FUNCTION "SSA_Analog_S5_to_S7" : VOID	// FC 109
TITLE = Scale S7 Analogues for S5
//COPYRIGHT:    (C) 1998 BY  BUHLER AG
//                           CH-9240 UZWIL  SWITZERLAND
//
//PRODUCT:      AME01_98
//
//TITLE:        Scale S7 Analogues for S5
//              
//
//-------------------------------------------------------------------------
//
//IDENT:        AUTHOR:             DEPT:             DATE:
//
//FC109.1A      GS                  CDDP              15-Jan-2000
//              1st Release
//
//-------------------------------------------------------------------------
//
//PURPOSE: 
//
//RESTRICTIONS: 
//
//-------------------------------------------------------------------------
//
//Functions
//=========
//
//AI_Type:
//   1= S5 Analogue Input 4..20mA
//   2= S5 Analogue Input 0..+-10V or 0.. +-20mA
//   3= S5 Analogue Input PT100
// 
//  11= S5 Analogue Output 4..20mA
//  12= S5 Analogue Output 0..+-10V or 0.. +-20mA
AUTHOR : GS
FAMILY : ASW
NAME : ANA_S5_S
VERSION : 1.0
VAR_INPUT
  AI_Type : INT ;	//S5 Signal:
END_VAR
VAR_TEMP
  Inputvalue : INT ;
  OutputValue : INT ;
END_VAR
BEGIN
NETWORK
TITLE = Initialisation
      TAK;
      T     #Inputvalue;
NETWORK
TITLE = S5 Analogue Input 4..20mA
// (network holds code this reader does not know; not shown)
// S5 Analogue inputs cards 4..20mA give a number of 0..2560
// but have an offset of 512. This gives 512..2560 = 4..20mA
// 2048 units cover 16mA.
// Bottom 3 bits are used for over/under range indication from the card
// All S7 modules use 0..27648 as 0..100%
// Conversion formula is:-
//  
//     (S5Value - 512)  * 27648
//     ---------------
//          2048
// 
NETWORK
TITLE = S5 Analogue Input: 0..+-10V , 0..+-20mA
// (network holds code this reader does not know; not shown)
// S5 Analogue inputs cards 0..20mA give a number of 0..2048
// Bottom 3 bits are used for over/under range indication from the card
// All S7 modules use 0..27648 as 0..100%
// Conversion formula is:-
//  
//     S5Value  * 27648
//     -------
//      2048
// 
NETWORK
TITLE = S5 Analogue Input: PT100
// (network holds code this reader does not know; not shown)
// S5 Analogue inputs cards 0..20mA give a number of 0..2048
// Bottom 3 bits are used for over/under range indication from the card
// All S7 modules use 0..27648 as 0..100%
// Conversion formula is:-
//  
//     (S5Value-1024)  * 27648
//     -------
//      1024
// 
NETWORK
TITLE = S5 Analogue Output 4..20mA
      L     #AI_Type;
      L     11;
      <>I;
      JC    M007;
// S5 Analogue Outputs cards use a number of 0..1024
// Bottom 4 bits are not used used
// All S7 modules use 0..27648 as 0..100%
// Conversion formula is:-
//  
//    ( S7Value  * 820 ) + 204
//      -------
//       27648
// 
// Note:   820 is 4/5ths of 1024    (for the 4..20mA portion)
//         204 is 1/5th of 1024     (for the 0..4mA portion)
// 
      L     #Inputvalue;
      DTR;
      L     2.764800e+04;	// 27648
      /R;
      L     8.200000e+02;	// 820
      *R;
      L     2.040000e+02;	// 204
      +R;
      RND;
      SLW   4;
      T     #OutputValue;
M007: NOP   0;
NETWORK
TITLE = S5 Analogue Output 0..20mA or 4..20mA card
      L     #AI_Type;
      L     12;
      <>I;
      JC    M008;
// S5 Analogue Outputs cards use a number of 0..1024
// Bottom 4 bits are not used used
// All S7 modules use 0..27648 as 0..100%
// Conversion formula is:-
//  
//     S7Value  * 1024
//     -------
//      27648
// 
      L     #Inputvalue;
      DTR;
      L     2.764800e+04;	// 27648
      /R;
      L     1.024000e+03;	// 1024
      *R;
      RND;
      SLW   4;
      T     #OutputValue;
M008: NOP   0;
NETWORK
TITLE = Output final value
      L     #OutputValue;
END_FUNCTION

FUNCTION "STD_LineSecStdSub" : VOID	// FC 120
TITLE = Line and section control standard subroutines
//COPYRIGHT:    (C) 2000 BY  BUHLER LTD.
//                           CH-9240 UZWIL  SWITZERLAND
//
//PRODUCT:      STD_MU664    
//
//TITLE:        Line and section control standard subroutines
//              
//              Standardfunktionen für Linien und Sektionen              
//              
//
//--------------------------------------------------------------------------------
//
//IDENT:        AUTOR:              DEPT:                              DATE:
//STD_FC120.2.0 A.Egli              CT3                                18-Oct-2002
//              - New release
//STD_FC120.1.12Ph. Engler          MU664                              23-Aug-2002
//              - Function (4,1) added: Search group manual mode
//STD_FC120.1.11Ph. Engler          MU664                              30-Apr-2002
//              - Function (1,55) and (2,55) modified: Stopping/Stopped
//STD_FC120.1.10Ph. Engler          MU664                              21-Mar-2002
//              - Function (2,55): starting until S.ToSSW.infStarted
//STD_FC120.1.9 Ph. Engler          MU664                              12-Mar-2002
//              Status codes for WinCoS implemented:
//              - General group colour code
//              - Line and Section info code
//STD_FC120.1.8 Ph. Engler          MU664                              20-Mar-2001
//              Line status colour for 2-4 section implemented
//STD_FC120.1.7 Ph. Engler          MU664                              20-Dec-2000
//              Pre stop weight for cmdSequenceStop
//STD_FC120.1.6 Ph. Engler          MU664                              14-Dec-2000
//              - Substitude Bincode into recipe extended, InCode 3 
//              - JS Job paramter flags (2,2) Sta-Address corrected
//STD_FC120.1.5 Ph. Engler          MU664                              01-Nov-2000
//              CmdSequenceStop only if section is in StActive           
//STD_FC120.1.4 Ph. Engler          MU664                              19-Okt-2000
//              Update SND-Binlist staSameSndRcv:
//               Suppression of the error meassage 'bin not found'
//STD_FC120.1.3 Ph. Engler          MU664                              28-Jun-2000
//              Section text and colour code extension 
//              with code 702, 703 and 1402
//STD_FC120.1.2 Ph. Engler          MU664                              04-May-2000
//              LS Line state/fault protocolling (1,10)
//               esXXX corrected 
//STD_FC120.1.1 Ph. Engler          MU664                              29-Mar-2000
//              Line log messages implemented
//STD_FC120.1.0 Ph. Engler          MU664                              05-Jan-2000
//              1st Release
//
//--------------------------------------------------------------------------------
//
//PURPOSE:      These function are callt by Line Control and
//              Section Control.
//              The most subroutine are handled by FB90
//
//RESTRICTIONS:
//
//--------------------------------------------------------------------------------
//
//InCode: 
//1000 to 1999: Subroutines Line
//              For Input and Output parameter is 
//              LineDB.VarTemp used  
//2000 to 2999: Subroutines Section
//              For Input and Output parameter is
//              SectionDB.VarTemp used  
//
//
//
//
AUTHOR : PE
FAMILY : STD
VERSION : 2.0
VAR_INPUT
  InCode : INT ;	//Code number; 1000=Line 2=Section
END_VAR
BEGIN
NETWORK
TITLE = Input Data
NETWORK
TITLE = Sub1031: CF Clear line flags 
//Open DB=  Line Parameter DB
      L     #InCode;
      L     1031;
      <>I;
      JC    CF00;
//Line parameter DB
      L     L#0;
      T     DBD 140;	// Section 1
      T     DBD 144;	// Section 2
      T     DBD 148;	// Section 3
      T     DBD 152;	// Section 4
      T     DBD 156;	// General
      T     DBD 160;	// General
CF00: NOP   0;
NETWORK
TITLE = All other Subroutines are handled by FB90
      CDB;
      L     #InCode;
      T     DIW 0;	//InCode
//Call Methode FB90
      UC    "STD_LineSecStdSub2";
END_FUNCTION

FUNCTION "ASW_StageCtrl_Fct" : VOID	// FC 1800
TITLE = Scale Control: Main routines
//COPYRIGHT:    (C) 1994 BY  BUHLER LTD.
//                           CH-9240 UZWIL  SWITZERLAND
//
//PRODUCT:      GCS7
//
//TITLE:        Stage Control
//
//Revision: 10
//
//-------------------------------------------------------------------------
//
//IDENT:        AUTOR:              DEPT:                         DATE:
//
//FC1800.1A     A.Egli              BSAE                          12.02.2008
//              Convert from S5 Version 2F
//
//-------------------------------------------------------------------------
//
//PURPOSE:      
//
//RESTRICTIONS:
//
//-------------------------------------------------------------------------
//
//FC-PARAMETER:
//------------
//InCode:
//
//   2= Init Batch
//   6= Next Stage
//
//  12= Init Stage
//      Update Stage.ScaleUsed
//      Stage.ScaleStarted:=0
//      Stage.ScaleDone
//
//
//  
AUTHOR : EA
FAMILY : GCS7UL
NAME : SCC_MAN
VERSION : 3.3
VAR_INPUT
  InCode : INT ;	// CODE
  Stage : UDT 18000;
END_VAR
VAR_TEMP
  tmpScaleDB : INT ;
  tmpScaleNr : DINT ;
  tmpScaleBit : DINT ;
  tmpRecipePlace : INT ;
  tmpRecipeDB : INT ;
  tmpRecipeAddrIngr : DINT ;
  tmpSecDB : INT ;
  tmpAddStage : DINT ;
  ConstMaxStage : INT ;
  tmpIdx : INT ;
  tmpOffsetIngr : INT ;	//Offest 1st Ingedient Stage [BYTE]
  tmpBinNo : INT ;
  tmpArrayIdxScale : INT ;
END_VAR
BEGIN
NETWORK
TITLE =
      L     2;
      T     #ConstMaxStage;
NETWORK
TITLE =
      L     P##Stage;
      LAR1;
      L     W [AR1,P#0.0];
      T     #tmpSecDB;
      L     D [AR1,P#2.0];
      T     #tmpAddStage;
NETWORK
TITLE = Call Section DB
      OPN   DB [#tmpSecDB];
      L     DBW 230;	// "SecDB".JobAc.RecipePlace
      T     #tmpRecipePlace;
NETWORK
TITLE = Methode 2: Init Batch
      L     #InCode;
      L     2;
      <>I;
      JC    iEnd;
      L     1;
      BLD   5;
      T     LD 36;	//--> Init Stage
      TAK;
      T     LD 40;
      L     P##Stage;
      LAR1;
      L     W [AR1,P#0.0];
      T     LW 34;
      OPN   DB [LW 34];
      L     D [AR1,P#2.0];
      LAR1;
      L     LD 40;
      L     LD 36;
      T     W [AR1,P#4.0];
      JU    dJ0;
iEnd: NOP   0;
NETWORK
TITLE = Methode 6: Next Stage
      L     #InCode;
      L     2;
      <>I;
      JC    nEnd;
      BLD   5;
      T     LD 36;
      TAK;
      T     LD 40;
      L     P##Stage;
      LAR1;
      L     W [AR1,P#0.0];
      T     LW 34;
      OPN   DB [LW 34];
      L     D [AR1,P#2.0];
      LAR1;
      L     LD 40;	//--> Init Stage
      L     LD 36;
      AN     [AR1,P#0.1];
      BLD   5;
      T     LD 36;
      TAK;
      T     LD 40;
      L     P##Stage;
      LAR1;
      L     W [AR1,P#0.0];
      T     LW 34;
      OPN   DB [LW 34];
      L     D [AR1,P#2.0];
      LAR1;
      L     LD 40;
      L     LD 36;
      AN     [AR1,P#2.0];
      BEC;
      L     #ConstMaxStage;
      BLD   5;
      T     LD 36;
      TAK;
      T     LD 40;
      L     P##Stage;
      LAR1;
      L     W [AR1,P#0.0];
      T     LW 34;
      OPN   DB [LW 34];
      L     D [AR1,P#2.0];
      LAR1;
      L     LD 40;
      L     LD 36;
      L     W [AR1,P#4.0];
      ==I;
      BLD   5;
      T     LD 36;
      TAK;
      T     LD 40;
      L     P##Stage;
      LAR1;
      L     W [AR1,P#0.0];
      T     LW 34;
      OPN   DB [LW 34];
      L     D [AR1,P#2.0];
      LAR1;
      L     LD 40;
      L     LD 36;
      S      [AR1,P#2.1];
      BEC;
      BLD   5;
      T     LD 36;
      TAK;
      T     LD 40;
      L     P##Stage;
      LAR1;
      L     W [AR1,P#0.0];
      T     LW 34;
      OPN   DB [LW 34];
      L     D [AR1,P#2.0];
      LAR1;
      L     LD 40;
      L     LD 36;
      L     W [AR1,P#4.0];
      +     1;
      BLD   5;
      T     LD 36;
      TAK;
      T     LD 40;
      L     P##Stage;
      LAR1;
      L     W [AR1,P#0.0];
      T     LW 34;
      OPN   DB [LW 34];
      L     D [AR1,P#2.0];
      LAR1;
      L     LD 40;
      L     LD 36;
      T     W [AR1,P#4.0];
      JU    dJ0;
nEnd: NOP   0;
NETWORK
TITLE = Methode 12: Init Stage
//ACTUAL DB BY CALL: Line DB
      L     #InCode;
      L     1;
      <>I;
      JC    dEnd;
//--------------------
//Init 
dJ0:  LAR1  #tmpAddStage;
      L     0;
      T     DBD [AR1,P#10.0];	//Stage.ScaleUsed
      T     DBD [AR1,P#14.0];	//Stage.ScaleUsed
      L     0;
      T     DBD [AR1,P#18.0];	//Stage.ScaleStarted
      T     DBD [AR1,P#22.0];	//Stage.ScaleStarted
      L     0;
      T     DBD [AR1,P#26.0];	//Stage.ScaleDone
      T     DBD [AR1,P#30.0];	//Stage.ScaleDone
      SET;
      BLD   5;
      T     LD 36;
      TAK;
      T     LD 40;
//Test Stage Number
      L     P##Stage;
      LAR1;
      L     W [AR1,P#0.0];
      T     LW 34;
      OPN   DB [LW 34];
      L     D [AR1,P#2.0];
      LAR1;
      L     LD 40;
//--------------------
//Loop over all In reipe used scales
      L     LD 36;
      R      [AR1,P#0.1];	//  
      BLD   5;
      T     LD 36;
      TAK;
      T     LD 40;	// "SecDB".JobNom.ScaleUsed[x]
      L     P##Stage;
      LAR1;
      L     W [AR1,P#0.0];
      T     LW 34;	//--> DB8.ScaleNr
      OPN   DB [LW 34];	// Subroutine ScalePointer
      L     D [AR1,P#2.0];
      LAR1;	//<--DB8.ScaleDB
      L     LD 40;
      L     LD 36;	// No Scale
      R      [AR1,P#0.0];
      BLD   5;
//--------------------
//Calculate Pointer to CWA Recipe
      T     LD 36;	// >>> CALL Scale-DB
      TAK;
      T     LD 40;
      L     P##Stage;
      LAR1;	// REC .ParNrOfIngrPerRecipe
      L     W [AR1,P#0.0];
      T     LW 34;
      OPN   DB [LW 34];
      L     D [AR1,P#2.0];
      LAR1;	// SCDB.ParNrOfBytePerIngr
      L     LD 40;	// 
      L     LD 36;	//---> Offset 1st Ingr. actual Stage
      R      [AR1,P#2.1];	// REC .ParNrOfIngrPerRecipe
      BLD   5;	// SCDB.ParNrOfBytePerIngr
      T     LD 36;	// 
      TAK;
      T     LD 40;	// 
      L     P##Stage;	// REC.ParDwNrFirstRecipe
      LAR1;	// --> Start Recipe[x]
      L     W [AR1,P#0.0];
      T     LW 34;
      OPN   DB [LW 34];
      L     D [AR1,P#2.0];	//-->Address Ingrediewnt 
      LAR1;
      L     LD 40;	// REC.ParDBNrRecipe
      L     LD 36;
//--------------------
//Read Ingredient from CWA recipe
      S      [AR1,P#2.0];	// >>> CALL Scale-DB
      BLD   5;
      T     LD 36;
//--------------------
//Set Scale Used
      TAK;
      T     LD 40;
      L     P##Stage;
      LAR1;	//--> not used
      L     W [AR1,P#0.0];
      T     LW 34;
      OPN   DB [LW 34];
      L     D [AR1,P#2.0];	//Stage.ScaleUsedStage
      LAR1;
      L     LD 40;
      L     LD 36;
      L     W [AR1,P#4.0];
      L     0;
//---------------------------------
//Test Stage Empty
      ==I;
      JC    dSta;
      BLD   5;
      T     LD 36;
      TAK;
      T     LD 40;
      L     P##Stage;
      LAR1;
      L     W [AR1,P#0.0];
      T     LW 34;
// -- END LOOP SCALE -----------
      OPN   DB [LW 34];
      L     D [AR1,P#2.0];
      LAR1;
      L     LD 40;
      L     LD 36;
      L     W [AR1,P#4.0];
      L     #ConstMaxStage;
      >I;
      JC    dSta;
      L     1;
dLPS: T     #tmpScaleNr;
      +     -1;
      T     #tmpArrayIdxScale;
      LAR1;
      AN    DBX [AR1,P#170.0];
      JC    dNxt;
      OPN   DI 8;
      L     #tmpScaleNr;
      T     DIW 20;
      CALL  "GCS7_ScaleCtrlSub" (
           CODE                     := 3);
      L     DIW 22;
      T     #tmpScaleDB;
      L     0;
      ==I;
      JC    dNxt;
      OPN   DI [#tmpScaleDB];
      BLD   5;
      T     LD 36;
      TAK;
      T     LD 40;
      L     P##Stage;
      LAR1;
      L     W [AR1,P#0.0];
      T     LW 34;
      OPN   DB [LW 34];
      L     D [AR1,P#2.0];
      LAR1;
      L     LD 40;
      L     LD 36;
      L     W [AR1,P#4.0];
      +     -1;
      T     #tmpIdx;
      L     DIW 104;
      L     #ConstMaxStage;
      /I;
      L     #tmpIdx;
      *I;
      L     DIW 106;
      *I;
      T     #tmpOffsetIngr;
      L     DIW 104;
      L     DIW 106;
      *I;
      L     #tmpRecipePlace;
      *I;
      L     DIW 100;
      +I;
      L     #tmpOffsetIngr;
      +D;
      SLD   3;
      T     #tmpRecipeAddrIngr;
      LAR1;
      L     DIW 98;
      T     #tmpRecipeDB;
      OPN   DI [#tmpRecipeDB];
      L     DIW [#tmpRecipeAddrIngr];
      T     #tmpBinNo;
      L     #tmpBinNo;
      L     0;
      ==I;
      JC    dNxt;
      LAR1  #tmpAddStage;
      L     #tmpArrayIdxScale;
      +AR1;
      S     DBX [AR1,P#10.0];
dNxt: L     64;
      L     #tmpScaleNr;
      +     1;
      >I;
      JC    dLPS;
dSta: LAR1  #tmpAddStage;
      L     DBD [AR1,P#10.0];
      L     0;
      ==D;
      A(;
      L     DBD [AR1,P#14.0];
      L     0;
      ==D;
      );
      BLD   5;
      T     LD 36;
      TAK;
      T     LD 40;
      L     P##Stage;
      LAR1;
      L     W [AR1,P#0.0];
      T     LW 34;
      OPN   DB [LW 34];
      L     D [AR1,P#2.0];
      LAR1;
      L     LD 40;
      L     LD 36;
      =      [AR1,P#2.0];
      BEU;
dEnd: NOP   0;
END_FUNCTION

FUNCTION "SSA_Vis_Update" : VOID	// FC 2042
TITLE = SSA_VIS_Status
//
//COPYRIGHT:    (C) 1996  BUHLER AG, CH-9240 UZWIL, SWITZERLAND
//
//PRODUCT:      SSA_VIS_Hsk
//
//TITLE:        Update hanshake bits for graphik update
//
//REVISION:     0
//-------------------------------------------------------------------------
//
//IDENT:        AUTHOR:             DEPT:                       DATE:
//FC2043.1.0    A. Egli             CT3                         19-Dec-2007
//              1st Release in S7
//
//-------------------------------------------------------------------------
//
//PURPOSE:      MANUAL : 
//
//RESTRICTIONS: S7
//-------------------------------------------------------------------------
//
FAMILY : ASW
NAME : SSA_VIS
VERSION : 1.0
VAR_INPUT
  HskDB : BLOCK_DB ;	//Pointer to Object Status
END_VAR
BEGIN
NETWORK
TITLE = Read Pointer
      OPN   #HskDB;
NETWORK
TITLE = Reset Handshake Bits
      NOP   0;
// Set Handshake Bit
      L     DBD 66;	// PCWrite_Graphic_Hsk
      INVD;	// 
      L     DBD 48;	// PCRead_Graphic_Hsk
      AD;	//  
      L     DBD 30;	// Graphic_Refresh
      OD;	// 
      T     DBD 48;	// PCRead_Graphic_Hsk
      L     DBD 70;	// PCWrite_Graphic_Hsk
      INVD;	// 
      L     DBD 52;	// PCRead_Graphic_Hsk
      AD;	//  
      L     DBD 34;	// Graphic_Refresh
      OD;	// 
      T     DBD 52;	// PCRead_Graphic_Hsk
      L     DBW 74;	// PCWrite_Graphic_Hsk
      INVI;	// 
      L     DBW 56;	// PCRead_Graphic_Hsk
      AW;	//  
      L     DBW 38;	// Graphic_Refresh
      OW;	// 
      T     DBW 56;	// PCRead_Graphic_Hsk
// Nachfrischen loeschen
      L     DBD 66;	//PCWrite_Graphic_Hsk
      INVD;
      L     DBD 30;	//Graphic_Refresh 
      AD;
      T     DBD 30;	//Graphic_Refresh
      L     DBD 70;	//PCWrite_Graphic_Hsk
      INVD;
      L     DBD 34;	//Graphic_Refresh 
      AD;
      T     DBD 34;	//Graphic_Refresh
      L     DBW 74;	//PCWrite_Graphic_Hsk
      INVI;
      L     DBW 38;	//Graphic_Refresh 
      AW;
      T     DBW 38;	//Graphic_Refresh
// Loeschen HS-Bit von VISCONTROL
      L     0;
      T     DBD 66;	//PCWrite_Graphic_Hsk
      T     DBD 70;	//PCWrite_Graphic_Hsk
      T     DBW 74;	//PCWrite_Graphic_Hsk
END_FUNCTION

FUNCTION "SSA_VIS_Status" : VOID	// FC 2043
TITLE = SSA_VIS_Status
//
//COPYRIGHT:    (C) 1996  BUHLER AG, CH-9240 UZWIL, SWITZERLAND
//
//PRODUCT:      SSA_VIS_Status
//
//TITLE:        Convert Status for Viscontrol
//
//REVISION:     0
//-------------------------------------------------------------------------
//
//IDENT:        AUTHOR:             DEPT:                       DATE:
//FC2043.1.0    A. Egli             CT3                         19-Dec-2007
//              1st Release in S7
//
//-------------------------------------------------------------------------
//
//PURPOSE:      MANUAL : 
//
//RESTRICTIONS: S7
//-------------------------------------------------------------------------
//
FAMILY : ASW
NAME : SSA_VIS
VERSION : 1.0
VAR_INPUT
  InObject : POINTER ;	//Pointer to Object Status
  OType : INT ;	//Object Type
  OutVisStatus : POINTER ;	//Pointer to Viscontrol Status in Picture DB
END_VAR
VAR_TEMP
  SrcDB : INT ;
  SrcAddress : DINT ;
  DstDB : INT ;
  DstAddress : DINT ;
  tmpDX : INT ;
END_VAR
BEGIN
NETWORK
TITLE = Read Pointer
      L     P##InObject;
      LAR1;
      L     W [AR1,P#0.0];
      T     #SrcDB;
      L     D [AR1,P#2.0];
      T     #SrcAddress;
      LAR2;
      OPN   DI [#SrcDB];
      L     P##OutVisStatus;
      LAR1;
      L     W [AR1,P#0.0];
      T     #DstDB;
      L     D [AR1,P#2.0];
      T     #DstAddress;
NETWORK
TITLE = Check Object Type
      L     1300;
      L     #OType;
      >=I;
      JC    ElMa;	//Element
      L     2300;
      L     #OType;
      >=I;
      JC    ElMa;	//Machine
      L     3000;
      L     #OType;
      ==I;
      JC    Gr;
      BEU;
NETWORK
TITLE =
ElMa: L     1000;
      /I;
      SRD   16;
      T     #tmpDX;
      JU    Calc;
NETWORK
TITLE =
Gr:   LAR2  P#DIX 0.0;
      A     DIX [AR2,P#21.4];	//Gr.OutWarning
      O     DIX [AR2,P#17.4];	//Gr.StFault
      L     2;
      JC    TRAN;
      O     DIX [AR2,P#17.2];	//Gr.StStarted
      O     DIX [AR2,P#17.3];	//Gr.StStopping
      L     1;
      JC    TRAN;
      O     DIX [AR2,P#17.0];	//Gr.StStopped
      O     DIX [AR2,P#17.1];	//Gr.StStarting
      L     0;
      JC    TRAN;
      L     99;
      JU    TRAN;
NETWORK
TITLE = Convert Status of ELement or Machine with Filter DB
Calc: NOP   0;
      L     123;
      L     #tmpDX;
      >I;
      JC    Err;
      L     249;
      L     #tmpDX;
      <I;
      JC    Err;
      +     -123;
      L     P#16.0;
      *D;
      L     P#20.0;
      +D;
      LAR1;
      OPN   "SSA_VIS_Filter";
//----------------------
//Test First Left Bytes without Status
      L     DBD [AR1,P#12.0];	//STATUS = 3
      L     DW#16#FFFFFF00;
      AD;
      L     DID [AR2,P#2.0];
      AD;
      JZ    STL2;
      L     3;
      JU    TRAN;
STL2: L     DBD [AR1,P#8.0];	//STATUS = 2
      L     DW#16#FFFFFF00;
      AD;
      L     DID [AR2,P#2.0];
      AD;
      JZ    STL1;
      L     2;
      JU    TRAN;
STL1: L     DBD [AR1,P#4.0];	//STATUS = 1
      L     DW#16#FFFFFF00;
      AD;
      L     DID [AR2,P#2.0];
      AD;
      JZ    STL0;
      L     1;
      JU    TRAN;
STL0: L     DBD [AR1,P#0.0];
      L     DW#16#FFFFFF00;
      AD;
      L     DID [AR2,P#2.0];
      AD;
      JZ    STR3;
      L     0;
      JU    TRAN;
//----------------------
//Test Right Bytes with Status
STR3: L     DBD [AR1,P#12.0];	//STATUS = 3
      L     DW#16#FF;
      AD;
      L     DID [AR2,P#2.0];
      AD;
      JZ    STR2;
      L     3;
      JU    TRAN;
STR2: L     DBD [AR1,P#8.0];	//STATUS = 2
      L     DW#16#FF;
      AD;
      L     DID [AR2,P#2.0];
      AD;
      JZ    STR1;
      L     2;
      JU    TRAN;
STR1: L     DBD [AR1,P#4.0];	//STATUS = 1
      L     DW#16#FF;
      AD;
      L     DID [AR2,P#2.0];
      AD;
      JZ    STR0;
      L     1;
      JU    TRAN;
STR0: L     DBD [AR1,P#0.0];	//STATUS = 0
      L     DW#16#FF;
      AD;
      L     DID [AR2,P#2.0];
      AD;
      JZ    Err;
      L     0;
      JU    TRAN;
Err:  L     99;	//Error
NETWORK
TITLE = Write Status to Picture DB
TRAN: OPN   DB [#DstDB];
      LAR1  #DstAddress;
      L     DBW [AR1,P#0.0];
      TAK;
      ==I;
      T     DBW [AR1,P#0.0];
      BEC;
//Set Change Bit
      L     #DstAddress;
      L     DW#16#FFFFF;
      AD;
      SRD   3;
      +     -2;
      L     "SSA_VIS_Filter".ParBlockLen;
      /I;
      L     2#1;
      SLW;
      OPN   DB [#DstDB];
      L     DBB 1;
      OW;
      T     DBB 1;
END_FUNCTION

FUNCTION "SSA_VIS_Log_Msg" : VOID	// FC 2055
TITLE = SSA_VIS_Log_Msg
//
//COPYRIGHT:    (C) 1996  BUHLER AG, CH-9240 UZWIL, SWITZERLAND
//
//PRODUCT:      GCS7R1
//
//TITLE:        LOG-TRANSFER FROM QUEUE TO VIS-VONTROL HANDSHAKE-DB
//
//REVISION:     0
//-------------------------------------------------------------------------
//
//IDENT:        AUTHOR:             DEPT:                       DATE:
//FC2055.1.0    A. Egli             CT3                         19-Dec-2007
//              1st Release in S7
//
//-------------------------------------------------------------------------
//
//PURPOSE:      MANUAL : 
//
//RESTRICTIONS: S7
//-------------------------------------------------------------------------
//
FAMILY : ASW
NAME : SSA_VIS
VERSION : 1.0
VAR_INPUT
  HSDB : BLOCK_DB ;	//VISCONTROL-HANDSHAKE-DB
  LogQueue : BLOCK_DB ;	//LOG-WARTESCHLANGE
  PCNr : INT ;	//UNTERSTUETZT WERDEN 2 PC's PCNR=1 und PCNR=2
  VDU : BOOL ;	//BITINFORMATION, OB VDU-MELDUNG ODER NICHT
END_VAR
VAR_TEMP
  tmpPC1 : BOOL ;
  tmpPC2 : BOOL ;
END_VAR
BEGIN
NETWORK
TITLE = Init
      L     #PCNr;
      L     1;
      ==I;
      =     #tmpPC1;	//PC 1
      L     #PCNr;
      L     2;
      ==I;
      =     #tmpPC2;	//PC 2
NETWORK
TITLE =
      OPN   #LogQueue;
      CDB;
      OPN   #HSDB;
NETWORK
TITLE = Reset Handshake LOG
      OPN   #HSDB;	// AUFRUF HSDB
      L     DBW 76;	// HSDB.PCWrite_LOG_Hsk   :  VIS->PLC:LOG-Daten gelesen
      INVI;	// 
      L     DBW 58;	// HSDB.PCRead_LOG_Hsk
      AW;
      T     DBW 58;	// HSDB.PCRead_LOG_Hsk    :  Reset Handshake Bits to PC
      L     0;
      T     DBW 76;	// HSDB.PCWrite_LOG_Hsk   :  Reset Handshake Bits from PC
NETWORK
TITLE = Enter Next Message
      AN    DIX 57.0;	//LogDB.HskPLCtoPC.PC1
      A     #tmpPC1;	//PC 1
      O;
      AN    DIX 57.1;	//LogDB.HskPLCtoPC.PC2
      A     #tmpPC2;	//PC 2
      O;
      A     DBX 59.0;	//HskDB.PCRead_LOG_Hsk 
      AN    #VDU;	//)  Element-Meldungen
      O;
      A     DBX 59.1;	//HskDB.PCRead_LOG_Hsk
      A     #VDU;	// VDU-Meldungen
      JC    END;
//Enter Next Message
      AN    #VDU;	// Element-Meldung
      JC    LOG;
      L     DIB 64;
      T     DBW 102;	// HskDB.Bildnummer
      S     DBX 59.1;	// HskDB.PCRead_LOG_Hsk.Bildnummer gueltig
      JU    RESE;
LOG:  L     DIW 60;	//)
      L     2#11111;	// )  LOG-HEAD KLASSE = 0
      AW;	// )
      L     16;	//)
      >=I;
      L     DIW 60;	// )
      JC    CWA;	// )
      L     2#1111111100011111;	// )  LOG-HEAD KLASSE = 0
      AW;	//  )
CWA:  T     DBW 78;	//-->HskDB.PCReadLog
      L     DIW 62;	// LogDB.PC.Msg[1]
      T     DBW 80;	//-->HskDB.PCReadLog
      L     DID 64;	// LogDB.PC.Msg[1]
      T     DBD 82;	//-->HskDB.PCReadLog
      L     DID 68;	// LogDB.PC.Msg[1]
      T     DBD 86;	//-->HskDB.PCReadLog
      L     DID 72;	// LogDB.PC.Msg[1]
      T     DBD 90;	//-->HskDB.PCReadLog
      L     DID 76;	// LogDB.PC.Msg[1]
      T     DBD 94;	//-->HskDB.PCReadLog
      L     DID 80;	// LogDB.PC.Msg[1]
      T     DBD 98;	//-->HskDB.PCReadLog
      SET;
      =     DBX 59.0;	//HskDB.PCRead_LOG_Hsk: Neue LOG-Daten!
//Set Message Done
RESE: A     #tmpPC1;	//PC1
      S     DIX 49.0;	//LogDB.PC.HskPC1toPLC 
      A     #tmpPC2;	//PC2
      S     DIX 51.0;	//LogDB.PC.HskPC2toPLC
END:  NOP   0;
END_FUNCTION

DATA_BLOCK "SYS_CBitDB"	// DB 2
TITLE = SYS: Changebit interface
//COPYRIGHT:    (C) 1994 BY  BUHLER LTD.
//                           CH-9240 UZWIL  SWITZERLAND
//
//PRODUCT:      GCS90
//
//TITLE:        Change-DB
//
//-------------------------------------------------------------------------
//
//IDENT:        AUTOR:              DEPT:                         DATE:
//
//DB250.1A      A.Egli              AEE61                         08-Jul-96
//                 1st Release
//
//-------------------------------------------------------------------------
//
//PURPOSE:      MANUAL : CBITMAN
//              CODE   : FB 74
//
//RESTRICTIONS:
//
//-------------------------------------------------------------------------
//
//$EJECT
//
//
//
//
AUTHOR : EA
FAMILY : GCS7SYS
NAME : CBIT_DB
VERSION : 0.0
  STRUCT
   Spare0 : WORD ;
   Spare2 : WORD ;
   Spare4 : WORD ;
   ParNextDB : INT ;	//Next Change-Bit DB
   Spare8 : WORD ;
   ParDWCopyBits : INT  := 512;	//Byte address of Copy[1]
   ParBlockLen : INT  := 120;	//Length datablock per change bit
   Spare14 : WORD ;
   Spare16 : WORD ;
   Spare18 : WORD ;
   VarTemp : ARRAY  [1 .. 10 ] OF //Working memory
   WORD ;
   RBit : ARRAY  [1 .. 1280 ] OF //-- PC Write ---------
   BOOL ;
   CBIT : ARRAY  [1 .. 1280 ] OF //-- PC Read  ------------
   BOOL ;
   Value : ARRAY  [1 .. 76 ] OF //Fast value for PC
   INT ;
   Copy : ARRAY  [1 .. 1280 ] OF //Internal used
   BOOL ;
   ParPointer : STRUCT 	//-- Configuaration source address --
    B001 : STRUCT
     DBNr : INT ;
     DWNr : INT ;
    END_STRUCT ;
    B005 : STRUCT
     DBNr : INT ;
     DWNr : INT ;
    END_STRUCT ;
    B009 : STRUCT
     DBNr : INT ;
     DWNr : INT ;
    END_STRUCT ;
    B013 : STRUCT
     DBNr : INT ;
     DWNr : INT ;
    END_STRUCT ;
    B017 : STRUCT
     DBNr : INT ;
     DWNr : INT ;
    END_STRUCT ;
    B021 : STRUCT
     DBNr : INT ;
     DWNr : INT ;
    END_STRUCT ;
    B025 : STRUCT
     DBNr : INT ;
     DWNr : INT ;
    END_STRUCT ;
    B029 : STRUCT
     DBNr : INT ;
     DWNr : INT ;
    END_STRUCT ;
    B033 : STRUCT
     DBNr : INT ;
     DWNr : INT ;
    END_STRUCT ;
    B037 : STRUCT
     DBNr : INT ;
     DWNr : INT ;
    END_STRUCT ;
    B041 : STRUCT
     DBNr : INT ;
     DWNr : INT ;
    END_STRUCT ;
    B045 : STRUCT
     DBNr : INT ;
     DWNr : INT ;
    END_STRUCT ;
    B049 : STRUCT
     DBNr : INT ;
     DWNr : INT ;
    END_STRUCT ;
    B053 : STRUCT
     DBNr : INT ;
     DWNr : INT ;
    END_STRUCT ;
    B057 : STRUCT
     DBNr : INT ;
     DWNr : INT ;
    END_STRUCT ;
    B061 : STRUCT
     DBNr : INT ;
     DWNr : INT ;
    END_STRUCT ;
    B065 : STRUCT
     DBNr : INT ;
     DWNr : INT ;
    END_STRUCT ;
    B069 : STRUCT
     DBNr : INT ;
     DWNr : INT ;
    END_STRUCT ;
    B073 : STRUCT
     DBNr : INT ;
     DWNr : INT ;
    END_STRUCT ;
    B077 : STRUCT
     DBNr : INT ;
     DWNr : INT ;
    END_STRUCT ;
    B081 : STRUCT
     DBNr : INT ;
     DWNr : INT ;
    END_STRUCT ;
    B085 : STRUCT
     DBNr : INT ;
     DWNr : INT ;
    END_STRUCT ;
    B089 : STRUCT
     DBNr : INT ;
     DWNr : INT ;
    END_STRUCT ;
    B093 : STRUCT
     DBNr : INT ;
     DWNr : INT ;
    END_STRUCT ;
    B097 : STRUCT
     DBNr : INT ;
     DWNr : INT ;
    END_STRUCT ;
    B101 : STRUCT
     DBNr : INT ;
     DWNr : INT ;
    END_STRUCT ;
    B105 : STRUCT
     DBNr : INT ;
     DWNr : INT ;
    END_STRUCT ;
    B109 : STRUCT
     DBNr : INT ;
     DWNr : INT ;
    END_STRUCT ;
    B113 : STRUCT
     DBNr : INT ;
     DWNr : INT ;
    END_STRUCT ;
    B117 : STRUCT
     DBNr : INT ;
     DWNr : INT ;
    END_STRUCT ;
    B121 : STRUCT
     DBNr : INT ;
     DWNr : INT ;
    END_STRUCT ;
   END_STRUCT ;
  END_STRUCT ;	
BEGIN
   ParDWCopyBits := 512;
   ParBlockLen := 120;
   ParPointer.B001.DBNr := -1;
END_DATA_BLOCK

DATA_BLOCK "SYS_DirectCtrlDB"	// DB 3
TITLE = GCS7: PC direct control interface default DB
AUTHOR : EA
FAMILY : GCS7SYS
NAME : PCCtrl
VERSION : 0.0
  STRUCT
   Spare0 : WORD ;
   Spare2 : WORD ;
   Spare4 : WORD ;
   Spare6 : DWORD ;
   Spare10 : DWORD ;
   ParAnswerTime : INT  := 5;	//Maximum time for answer
   VarActControlDB : INT ;	//DB from actual communication
   VarAnswerTime : INT ;	//Actual answer time
   GC : STRUCT 	//=== Working memory
    InDBNr : INT ;
    InDynLen : INT ;
    InDynAddr : DINT ;
    InParaLen : INT ;
    InParaAddr : DINT ;
    Revision : INT ;
    Temp8 : DINT ;
   END_STRUCT ;
   ChangeBit : STRUCT 	//Change Bit
    Spare : BYTE ;
    CBit1 : BOOL ;	//Function done
    CBit2 : BOOL ;
    CBit3 : BOOL ;
    CBit4 : BOOL ;
   END_STRUCT ;
   PC : STRUCT 	//== PC: Read/Write
    Hsk : STRUCT 	// Handshake
     Spare0 : BYTE ;
     FDefineCmd : BOOL ;
     FDefinePara : BOOL ;
     FDefineValue : BOOL ;
     FExamine : BOOL ;
     F04 : BOOL ;
     F05 : BOOL ;
     F06 : BOOL ;
     F07 : BOOL ;
    END_STRUCT ;
    ErrObj : INT ;	//Spare
    ErrCode : INT ;	//Fault reason: 0=No Fault
    ObjectType : INT ;	//Type of addressed object
    ObjectNo : INT ;	//Addressd object
    Cmd1 : ARRAY  [0 .. 15 ] OF BOOL ;
    Cmd2 : ARRAY  [0 .. 15 ] OF BOOL ;
    Cmd3 : ARRAY  [0 .. 15 ] OF BOOL ;
    Value : ARRAY  [1 .. 100 ] OF //Data from or for actual object
    WORD ;
   END_STRUCT ;
  END_STRUCT ;	
BEGIN
   ParAnswerTime := 5;
END_DATA_BLOCK

DATA_BLOCK "SYS_HornDB"	// DB 4
TITLE = GCS7: Data Horn Modul
//COPYRIGHT:    (C) 2000 BUHLER AG, CH-9240 UZWIL, SWITZERLAND
//                           
//PRODUCT:      Horn DB
//              Horn DB
//
//TITLE:        Horn Modul
//              
//
//--------------------------------------------------------------------------------
//
//IDENT:        AUTHOR:             DEPT:                              DATE:
//
//P01_DB004.2.0 A_Egli              CT3                                29.Okt.2002
//              1st Release
//
//-------------------------------------------------------------------------
//
AUTHOR : EA
FAMILY : GCSS7
NAME : HornDB
VERSION : 2.0
  STRUCT
   All : STRUCT
    CmdHornOff : BOOL ;
    Spare1 : BOOL ;
    Spare2 : BOOL ;
    Spare3 : BOOL ;
    Spare4 : BOOL ;
    Spare5 : BOOL ;
   END_STRUCT ;
   _1_A901Horn : STRUCT
    CmdHornOff : BOOL ;
    CmdHornOn : BOOL ;
    StartWarning : BOOL ;
    Spare1 : BOOL ;
    Spare2 : BOOL ;
   END_STRUCT ;
   _1_A902Horn : STRUCT
    CmdHornOff : BOOL ;
    CmdHornOn : BOOL ;
    StartWarning : BOOL ;
    Spare1 : BOOL ;
    Spare2 : BOOL ;
   END_STRUCT ;
   _1_A903Horn : STRUCT
    CmdHornOff : BOOL ;
    CmdHornOn : BOOL ;
    StartWarning : BOOL ;
    Spare1 : BOOL ;
    Spare2 : BOOL ;
   END_STRUCT ;
   _1_A904Horn : STRUCT
    CmdHornOff : BOOL ;
    CmdHornOn : BOOL ;
    StartWarning : BOOL ;
    Spare1 : BOOL ;
    Spare2 : BOOL ;
   END_STRUCT ;
  END_STRUCT ;	
BEGIN
END_DATA_BLOCK

DATA_BLOCK "SYS_LOG_Queue"	// DB 5
TITLE = SYS_LOG_Queue
//COPYRIGHT:    (C) 1996 BY  BUHLER LTD.
//                           CH-9240 UZWIL  SWITZERLAND
//
//PRODUCT:      GCS90_OS.LOG
//
//TITLE:        QUEUE-DB
//
//-------------------------------------------------------------------------
//
//IDENT:        AUTOR:              DEPT:                       DATE:
//
//DB5.1A        S. Kalberer         AEE61                       4-Jun-1996
//              1st Release in S7, converted from DB220.1A
//
//-------------------------------------------------------------------------
//
//PURPOSE:      MANUAL : LOGMAN
//              CODE   : FB46,47
//
//RESTRICTIONS: S7
//              only for PC-Interface
//
//-------------------------------------------------------------------------
//
//
AUTHOR : SK
FAMILY : GCS7SYS
NAME : LOG_DB
VERSION : 0.0
  STRUCT
   spare0 : WORD ;
   ParByteStartQueue : INT  := 180;	//1st Byte of ParMsgQueue
   spare4 : INT ;
   ParMaxNoOfMsg : INT  := 100;	//Max index of array MsgQueue
   VarNrOfMsgInQueue : INT ;	//Actual number of Msg in queue
   VarByteWrite : INT ;	//Write pointer
   VarByteRead : INT ;	//Read pointer
   ParByteMsgFull : INT  := 156;	//1st Byte or ParMsgFull
   varMsg : STRUCT 	//== Working memory
    Header : WORD ;
    Para1 : WORD ;
    Para2 : WORD ;
    Para3 : WORD ;
    Para4 : WORD ;
    Para5 : WORD ;
    Para6 : WORD ;
    Para7 : WORD ;
    Para8 : WORD ;
    Para9 : WORD ;
    Para10 : WORD ;
    Para11 : WORD ;
   END_STRUCT ;
   ChangeBit : STRUCT
    spare : BYTE ;
    CBit0 : BOOL ;
   END_STRUCT ;
   ParNrOfMsgMemory : INT  := 1;	//Max index of array PC.Msg
   spare : BYTE ;
   ParPC1Connected : BOOL  := TRUE;	//Pc1 is connected
   ParPC2Connected : BOOL ;	//Pc1 is connected
   ParPC3Connected : BOOL ;	//Pc1 is connected
   ParPC4Connected : BOOL ;	//Pc1 is connected
   spare4504 : BOOL ;
   spare4505 : BOOL ;
   spare4506 : BOOL ;
   spare4507 : BOOL ;
   spare4600 : BOOL ;
   spare4601 : BOOL ;
   spare4602 : BOOL ;
   spare4603 : BOOL ;
   spare4604 : BOOL ;
   spare4605 : BOOL ;
   CmdAddFastMsg : BOOL ;	//->Add Fast Message directly at PC interface
   CmdResetLog : BOOL  := TRUE;	//->Init Queue
   InPC1Online : BOOL ;	//->PC1 is offline
   InPC2Online : BOOL ;	//->PC2 is offline
   InPC3Online : BOOL ;	//->PC3 is offline
   InPC4Online : BOOL ;	//->PC4 is offline
   PC : STRUCT 	//=== Interface to PC
    HskPC1toPLC : WORD ;
    HskPC2toPLC : WORD ;
    HskPC3toPLC : WORD ;
    HskPC4toPLC : WORD ;
    HskPLCtoPC : WORD ;
    NrOfMessageInQueue : WORD ;
    Msg : ARRAY  [1 .. 4 ] OF //Message for PC
    STRUCT
     Header : WORD ;
     Para1 : WORD ;
     Para2 : WORD ;
     Para3 : WORD ;
     Para4 : WORD ;
     Para5 : WORD ;
     Para6 : WORD ;
     Para7 : WORD ;
     Para8 : WORD ;
     Para9 : WORD ;
     Para10 : WORD ;
     Para11 : WORD ;
    END_STRUCT ;
   END_STRUCT ;
   ParMsgFull : STRUCT 	//===Message queue full
    Header : WORD  := W#16#8C;
    Para1 : WORD ;
    Para2 : WORD ;
    Para3 : WORD ;
    Para4 : WORD ;
    Para5 : WORD ;
    Para6 : WORD ;
    Para7 : WORD ;
    Para8 : WORD ;
    Para9 : WORD ;
    Para10 : WORD ;
    Para11 : WORD  := W#16#B;
   END_STRUCT ;
   MsgQueue : ARRAY  [1 .. 100 ] OF //=== Message buffer =========
   STRUCT
    Header : WORD ;
    Para1 : WORD ;
    Para2 : WORD ;
    Para3 : WORD ;
    Para4 : WORD ;
    Para5 : WORD ;
    Para6 : WORD ;
    Para7 : WORD ;
    Para8 : WORD ;
    Para9 : WORD ;
    Para10 : WORD ;
    Para11 : WORD ;
   END_STRUCT ;
  END_STRUCT ;	
BEGIN
   ParByteStartQueue := 180;
   ParMaxNoOfMsg := 100;
   ParByteMsgFull := 156;
   ParNrOfMsgMemory := 1;
   ParPC1Connected := TRUE;
   CmdResetLog := TRUE;
   ParMsgFull.Header := W#16#8C;
   ParMsgFull.Para11 := W#16#B;
END_DATA_BLOCK

DATA_BLOCK "GCS7_GrCtrlDBTmp"	// DB 6
AUTHOR : EA
FAMILY : GCS7UL
VERSION : 0.0
"GCS7_GrpCtrlMain"
BEGIN
END_DATA_BLOCK

DATA_BLOCK "GCS7_ScaleControlDB"	// DB 8
TITLE = GCS7_ScaleControlDB: Data of Scale Control modul
//
//COPYRIGHT:    (C) 1994 BY  BUHLER LTD.
//                           CH-9240 UZWIL  SWITZERLAND
//
//PRODUCT:      GCS90
//
//TITLE:        SCALE-CONTROL
//
//-------------------------------------------------------------------------
//
//IDENT:       AUTOR:              DEPT:             DATE:
//
//DB8.1A        A_Egli              AEE61             21.11.96
//              1st Release
//
//-------------------------------------------------------------------------
//
//PURPOSE:      MANUAL : SCCMAN
//              CODE   : FC68/FC69...
//
//RESTRICTIONS:
//
//-------------------------------------------------------------------------
//
//
AUTHOR : EA
FAMILY : GCS90UL
NAME : SCC_DB
VERSION : 0.0
  STRUCT
   spare0 : ARRAY  [0 .. 9 ] OF // reserved for parameter
   WORD ;
   VarTemp : ARRAY  [1 .. 11 ] OF // working memory
   WORD ;
   ParScaleDB : ARRAY  [1 .. 64 ] OF // Configuration of all scale DB
   INT ;
  END_STRUCT ;	
BEGIN
   ParScaleDB[1] := 201;
   ParScaleDB[2] := 202;
END_DATA_BLOCK

DATA_BLOCK "GCS7_GrCtrlDB"	// DB 9
TITLE = GCS7: Inteface Group to Group control
//COPYRIGHT:    (C) 2000 BUHLER AG, CH-9240 UZWIL, SWITZERLAND
//                           
//PRODUCT:      Gruppenverwaltung mit 320 Gruppen
//              Group Control with 320 groups
//
//TITLE:        Call Group FB
//              
//
//--------------------------------------------------------------------------------
//
//IDENT:        AUTHOR:             DEPT:                              DATE:
//
//P01_DB009.2.0 A_Egli              CT3                                31.Okt.2002
//              1st Release
//
//-------------------------------------------------------------------------
//
AUTHOR : EA
FAMILY : GCSS7
NAME : ObjDB
VERSION : 2.0
  STRUCT
   ParByteNoSecDB : INT  := 1012;	//Pointer to configuration of section DBs
   ParMaxGroupCnt : INT  := 10;	//1=32 Groups, 2=64 Groups,.. , 10= 320 Groups,
   OutManualAny : BOOL ;	//Any object of the plant in manual mode
   OutFaultAny : BOOL ;	//Any object of the plant has faull
   Spare4 : WORD ;
   Spare5 : WORD ;
   ParFeed : ARRAY  [1 .. 320 ] OF //Objects are feed groups
   BOOL ;
   ParMGR : ARRAY  [1 .. 320 ] OF //Objects are MGR
   BOOL ;
   ParWGR : ARRAY  [1 .. 320 ] OF //Objects are WGR
   BOOL ;
   ParGGR : ARRAY  [1 .. 320 ] OF //Objects are GGR
   BOOL ;
   ParShare : ARRAY  [1 .. 320 ] OF //Objects are possible to share
   BOOL ;
   OutShared : ARRAY  [1 .. 320 ] OF //Objects are shared at the moment
   BOOL ;
   OutOccupied : ARRAY  [1 .. 320 ] OF //Objects are occupied by any section
   BOOL ;
   OutEnable : ARRAY  [1 .. 320 ] OF //Enable for objects
   BOOL ;
   CmdNext : ARRAY  [1 .. 320 ] OF //Next command for objects
   BOOL ;
   CmdFaultReset : ARRAY  [1 .. 320 ] OF BOOL ;
   CmdManualOff : ARRAY  [1 .. 320 ] OF BOOL ;
   InStopped : ARRAY  [1 .. 320 ] OF BOOL ;
   InStarted : ARRAY  [1 .. 320 ] OF BOOL ;
   InFault : ARRAY  [1 .. 320 ] OF BOOL ;
   InWarning : ARRAY  [1 .. 320 ] OF BOOL ;
   InManual : ARRAY  [1 .. 320 ] OF BOOL ;
   InLocked : ARRAY  [1 .. 320 ] OF //Waiting until real group
   BOOL ;
   InExternal : ARRAY  [1 .. 320 ] OF //Is at the moment external used
   BOOL ;
   CmdContinue : ARRAY  [1 .. 320 ] OF //Is used as condition to set OutAutoStart
   BOOL ;
   InLoaded : ARRAY  [1 .. 320 ] OF //Group is loaded with product
   BOOL ;
   InDPFault : ARRAY  [1 .. 320 ] OF //Any element has DPFault
   BOOL ;
   InHWStop : ARRAY  [1 .. 320 ] OF //Any element has HWStop
   BOOL ;
   InAutoStart : ARRAY  [1 .. 320 ] OF //OutAutoStart is on
   BOOL ;
   InStartWarning : ARRAY  [1 .. 320 ] OF //InStartWarning is on
   BOOL ;
   OutConflictObj : ARRAY  [1 .. 320 ] OF BOOL ;
   OutConflictSecDB : INT ;
   Section : ARRAY  [1 .. 100 ] OF STRUCT
    DBNr : INT ;
    DBB : INT ;
   END_STRUCT ;
  END_STRUCT ;	
BEGIN
   ParByteNoSecDB := 1012;
   ParMaxGroupCnt := 10;
   ParFeed[26] := TRUE;
   ParFeed[33] := TRUE;
   ParFeed[41] := TRUE;
   ParFeed[43] := TRUE;
   ParFeed[46] := TRUE;
   ParMGR[22] := TRUE;
   ParMGR[24] := TRUE;
   ParMGR[31] := TRUE;
   ParMGR[32] := TRUE;
   ParMGR[42] := TRUE;
   ParMGR[44] := TRUE;
   ParMGR[45] := TRUE;
   ParMGR[47] := TRUE;
   ParMGR[196] := TRUE;
   ParWGR[12] := TRUE;
   ParWGR[13] := TRUE;
   ParWGR[21] := TRUE;
   ParWGR[23] := TRUE;
   ParWGR[28] := TRUE;
   ParGGR[1] := TRUE;
   ParGGR[2] := TRUE;
   ParGGR[7] := TRUE;
   ParShare[1] := TRUE;
   ParShare[2] := TRUE;
   ParShare[7] := TRUE;
END_DATA_BLOCK

DATA_BLOCK "SYS_DirectCtrlLCDB"	// DB 10
TITLE = GCS7: PC direct control interface default DB
AUTHOR : EA
FAMILY : GCS7SYS
NAME : PCCtrl
VERSION : 0.0
  STRUCT
   Spare0 : WORD ;
   Spare2 : WORD ;
   Spare4 : WORD ;
   Spare6 : DWORD ;
   Spare10 : DWORD ;
   ParAnswerTime : INT  := 10;	//Maximum time for answer
   VarActControlDB : INT ;	//DB from actual communication
   VarAnswerTime : INT ;	//Actual answer time
   GC : STRUCT 	//=== Working memory
    InDBNr : INT ;
    InDynLen : INT ;
    InDynAddr : DINT ;
    InParaLen : INT ;
    InParaAddr : DINT ;
    Set11Done : BOOL ;
    InObjectNo : INT ;
    InLCAddr : INT ;
   END_STRUCT ;
   ChangeBit : STRUCT 	//Change Bit
    Spare : BYTE ;
    CBit1 : BOOL ;	//Function done
    CBit2 : BOOL ;
    CBit3 : BOOL ;
    CBit4 : BOOL ;
   END_STRUCT ;
   PC : STRUCT 	//== PC: Read/Write
    Hsk : STRUCT 	// Handshake
     Spare0 : BYTE ;
     FDefineCmd : BOOL ;
     FDefinePara : BOOL ;
     FDefineValue : BOOL ;
     FExamine : BOOL ;
     FExamineFirst : BOOL ;
     FExamineNext : BOOL ;
     F06 : BOOL ;
     F07 : BOOL ;
    END_STRUCT ;
    ErrObj : INT ;	//Spare
    ErrCode : INT ;	//Fault reason: 0=No Fault
    ObjectType : INT ;	//Type of addressed object
    ObjectNo : INT ;	//Addressd object
    Cmd1 : ARRAY  [0 .. 15 ] OF BOOL ;
    Cmd2 : ARRAY  [0 .. 15 ] OF BOOL ;
    Cmd3 : ARRAY  [0 .. 15 ] OF BOOL ;
    Value : ARRAY  [1 .. 100 ] OF //Data from or for actual object
    WORD ;
   END_STRUCT ;
  END_STRUCT ;	
BEGIN
   ParAnswerTime := 10;
END_DATA_BLOCK

DATA_BLOCK "TEST_IOSimuliInput"	// DB 16
AUTHOR : EA
FAMILY : SIM
NAME : Inputs
VERSION : 0.1
  STRUCT
   in : ARRAY  [0 .. 1027 ] OF BYTE ;
  END_STRUCT ;	
BEGIN
END_DATA_BLOCK

DATA_BLOCK "TEST_IOSimuliOutput"	// DB 17
AUTHOR : EA
FAMILY : SIM
NAME : Inputs
VERSION : 0.1
  STRUCT
   in : ARRAY  [0 .. 1027 ] OF BYTE ;
  END_STRUCT ;	
BEGIN
END_DATA_BLOCK

DATA_BLOCK "KebaHT4Data"	// DB 20
AUTHOR : SK
FAMILY : KebaHT4
VERSION : 0.0
"KebaHT4"
BEGIN
END_DATA_BLOCK

DATA_BLOCK DB 21
TITLE = Reference List Motors for HT4 Control
//COPYRIGHT:    (C) 1999 BY  BUHLER LTD.
//                           CH-9240 UZWIL  SWITZERLAND
//
//PRODUCT:      
//
//TITLE:        REFERENCE LIST "MOTORS" FOR "MAINTENANCE MOTOR CONTROL HT4"
//
//              REFERENZLISTE "MOTOREN" FUER "LOKALE MOTOREN STEUERUNG HT4"
//
//---------------------------------------------------------------------------
//
//IDENT:        AUTHOR:              DEPT:                       DATE:
//
//DB81.1A       S. Kalberer          CT3                         14.04.1999
//              1st Release: adjusted from S5 DB181.2A
//
//---------------------------------------------------------------------------
//
//PURPOSE:      - REFERENCE TABLE FOR MOTOR ELEMENTS
//
//RESTRICTIONS: - S7
//              - THIS DB IS CALLED BY FB80.
//
//---------------------------------------------------------------------------
//
//STRUCTURE OF DB-BLOCKS:
//=======================
//Byte 00: DBW (WORD-Hex) = OBJECT No. (Motors with two direction/speed are marked with *)
//                                     (Motors with variable speed are marked with @)
//Byte 02: DBW (INT)  = Digital output 1 byte-address 
//Byte 04: DBW (INT)  = Digital output 1 bit-address
//Byte 06: DBW (INT)  = Digital output 2 byte-address 
//Byte 08: DBW (INT)  = Digital output 2 bit-address
//Byte 10: DBW (INT)  = Digital output 3 byte-address 
//Byte 12: DBW (INT)  = Digital output 3 bit-address
//Byte 14: DBW (INT)  = Digital output 4 byte-address 
//Byte 16: DBW (INT)  = Digital output 4 bit-address
//Byte 18: DBW (INT)  = Analog  output 1 address (byte)
//Byte 20: DBW (WORD) = Object  state
//
//PARAMETERS FOR OUTPUTS:
//=======================
//Motor: (with one direction or speed)
//DO_1 = Digital output address
//DO_2 = not used
//DO_3 = not used
//DO_4 = not used
//AO_1 = not used
//
//Motor: (with two directions or speed) *
//DO_1 = Digital output address (foreward/1.speed)
//DO_2 = Digital output address (reverse/2.speed)
//DO_3 = not used
//DO_4 = not used
//AO_1 = not used
//
//Motor: (with variable speed drive) @
//DO_1 = Digital output address
//DO_2 = not used
//DO_3 = not used
//DO_4 = not used
//AO_1 = Analog output address
//
//KNOW_HOW_PROTECT
// (falls angegeben, kann im generierten Baustein keine Änderungen mehr vorgenommen werden)
// (If specified, no more changes can be made once the block is generated)
//UNLINKED
// (falls angegeben, ist der generierte Baustein nur im AG Ladespeicher vorhanden) 
// (If specified, the generated block is only available in the PLC load memory)
//READ_ONLY
// (falls angegeben, ist der generierte Baustein im AG nicht änderbar)
// (If specified, the generated block cannot be changed in the programmable controller)
//
AUTHOR : ASW
FAMILY : Keba
NAME : DB_MOT
VERSION : 1.0
  STRUCT
   Obj : ARRAY  [1 .. 11 ] OF STRUCT
    No : WORD ;	//Object No. (e.g. 1002 for 1-M002)
    DO1_ByteAddr : INT ;	//DO1 (Byte Address)
    DO1_BitAddr : INT ;	//DO1 (Bit Address)
    DO2_ByteAddr : INT ;	//DO2 (Byte Address)
    DO2_BitAddr : INT ;	//DO2 (Bit Address)
    DO3_ByteAddr : INT ;	//DO3 (Byte Address)
    DO3_BitAddr : INT ;	//DO3 (Bit Address)
    DO4_ByteAddr : INT ;	//DO4 (Byte Address)
    DO4_BitAddr : INT ;	//DO4 (Bit Address)
    AO1_ByteAddr : INT ;	//AO1 (Byte Address)
    State : WORD ;	//State
   END_STRUCT ;
  END_STRUCT ;	
BEGIN
   Obj[1].No := W#16#1001;
   Obj[1].DO1_ByteAddr := 4;
   Obj[2].No := W#16#1002;
   Obj[2].DO1_ByteAddr := 4;
   Obj[2].DO1_BitAddr := 1;
   Obj[3].No := W#16#1003;
   Obj[3].DO1_ByteAddr := 4;
   Obj[3].DO1_BitAddr := 2;
   Obj[3].DO2_ByteAddr := 5;
   Obj[3].DO2_BitAddr := 2;
   Obj[4].No := W#16#1004;
   Obj[4].DO1_ByteAddr := 4;
   Obj[4].DO1_BitAddr := 3;
   Obj[4].DO2_ByteAddr := 5;
   Obj[4].DO2_BitAddr := 3;
   Obj[9].No := W#16#1010;
   Obj[9].DO1_ByteAddr := 4;
   Obj[9].DO1_BitAddr := 7;
   Obj[9].AO1_ByteAddr := 512;
   Obj[10].No := W#16#1011;
   Obj[10].DO1_ByteAddr := 5;
   Obj[10].AO1_ByteAddr := 20;
   Obj[11].No := W#16#FFFF;
END_DATA_BLOCK

DATA_BLOCK DB 22
TITLE = Reference List various Objects for HT4 Control
//COPYRIGHT:    (C) 1999 BY  BUHLER LTD.
//                           CH-9240 UZWIL  SWITZERLAND
//
//PRODUCT:      
//
//TITLE:        REFERENCE LIST "OBJECTS" FOR "MAINTENANCE MOTOR CONTROL HT4"
//
//              REFERENZLISTE "OBJEKTE" FUER "LOKALE MOTOREN STEUERUNG HT4"
//
//---------------------------------------------------------------------------
//
//IDENT:        AUTHOR:              DEPT:                       DATE:
//
//DB82.1A       S. Kalberer          CT3                         14.04.1999
//              1st Release: adjusted from S5 DB182.2A
//
//---------------------------------------------------------------------------
//
//PURPOSE:      - REFERENCE TABLE FOR VARIOUS ELEMENTS
//
//RESTRICTIONS: - S7
//              - THIS DB IS CALLED BY FB80.
//
//---------------------------------------------------------------------------
//
//STRUCTURE OF DB-BLOCKS:
//=======================
//Byte 00: DBW (WORD-Hex) = OBJECT No. (Motors with two direction/speed are marked with *)
//                                     (Motors with variable speed are marked with @)
//Byte 02: DBW (INT)  = Digital output 1 byte-address 
//Byte 04: DBW (INT)  = Digital output 1 bit-address
//Byte 06: DBW (INT)  = Digital output 2 byte-address 
//Byte 08: DBW (INT)  = Digital output 2 bit-address
//Byte 10: DBW (INT)  = Digital output 3 byte-address 
//Byte 12: DBW (INT)  = Digital output 3 bit-address
//Byte 14: DBW (INT)  = Digital output 4 byte-address 
//Byte 16: DBW (INT)  = Digital output 4 bit-address
//Byte 18: DBW (INT)  = Analog  output 1 address (byte)
//Byte 20: DBW (WORD) = Object  state
//
//
//PARAMETERS FOR OUTPUTS:
//=======================
//Motor: (with one direction or speed)
//DO_1 = Digital output address
//DO_2 = not used
//DO_3 = not used
//DO_4 = not used
//AO_1 = not used
//
//Motor: (with two directions or speed)
//DO_1 = Digital output address (foreward/1.speed)
//DO_2 = Digital output address (reverse/2.speed)
//DO_3 = not used
//DO_4 = not used
//AO_1 = not used
//
//Motor: (with variable speed drive)
//DO_1 = Digital output address
//DO_2 = not used
//DO_3 = not used
//DO_4 = not used
//AO_1 = Analog output address
//
//Valve: (double acting)
//DO_1 = LN (low number)
//DO_2 = HN (high number)
//DO_3 = not used
//DO_4 = not used
//AO_1 = not used
//
//Valve: (single acting)
//DO_1 = OFF
//DO_2 = ON
//DO_3 = not used
//DO_4 = not used
//AO_1 = not used
//
//Filter control Units:
//DO_1 = OFF
//DO_2 = ON
//DO_3 = not used
//DO_4 = not used
//AO_1 = not used
//KNOW_HOW_PROTECT
// (falls angegeben, kann im generierten Baustein keine Änderungen mehr vorgenommen werden)
// (If specified, no more changes can be made once the block is generated)
//UNLINKED
// (falls angegeben, ist der generierte Baustein nur im AG Ladespeicher vorhanden) 
// (If specified, the generated block is only available in the PLC load memory)
//READ_ONLY
// (falls angegeben, ist der generierte Baustein im AG nicht änderbar)
// (If specified, the generated block cannot be changed in the programmable controller)
//
AUTHOR : ASW
FAMILY : Keba
NAME : DB_Div
VERSION : 1.0
  STRUCT
   Obj : ARRAY  [1 .. 11 ] OF STRUCT
    No : WORD ;	//Object No. (e.g. 1417 for 1-417/418V)
    DO1_ByteAddr : INT ;	//DO1 (Byte Address)
    DO1_BitAddr : INT ;	//DO1 (Bit Address)
    DO2_ByteAddr : INT ;	//DO2 (Byte Address)
    DO2_BitAddr : INT ;	//DO2 (Bit Address)
    DO3_ByteAddr : INT ;	//DO3 (Byte Address)
    DO3_BitAddr : INT ;	//DO3 (Bit Address)
    DO4_ByteAddr : INT ;	//DO4 (Byte Address)
    DO4_BitAddr : INT ;	//DO4 (Bit Address)
    AO1_ByteAddr : INT ;	//AO1 (Byte Address)
    State : WORD ;	//State
   END_STRUCT ;
  END_STRUCT ;	
BEGIN
   Obj[1].No := W#16#1417;
   Obj[1].DO1_ByteAddr := 10;
   Obj[1].DO2_ByteAddr := 10;
   Obj[1].DO2_BitAddr := 1;
   Obj[2].No := W#16#1419;
   Obj[2].DO1_ByteAddr := 10;
   Obj[2].DO1_BitAddr := 2;
   Obj[2].DO2_ByteAddr := 10;
   Obj[2].DO2_BitAddr := 3;
   Obj[3].No := W#16#1003;
   Obj[3].DO1_ByteAddr := 4;
   Obj[3].DO1_BitAddr := 2;
   Obj[3].DO2_ByteAddr := 5;
   Obj[3].DO2_BitAddr := 2;
   Obj[4].No := W#16#1004;
   Obj[4].DO1_ByteAddr := 4;
   Obj[4].DO1_BitAddr := 3;
   Obj[4].DO2_ByteAddr := 5;
   Obj[4].DO2_BitAddr := 3;
   Obj[10].No := W#16#1011;
   Obj[10].DO1_ByteAddr := 5;
   Obj[10].DO1_BitAddr := 1;
   Obj[11].No := W#16#FFFF;
END_DATA_BLOCK

DATA_BLOCK "PLC_SystemDB"	// DB 50
TITLE = PLC: System informations
//COPYRIGHT:    (C) 2000 BY  BUHLER AG
//                           CH-9240 UZWIL  SWITZERLAND
//
//PRODUCT:      STD_MU664
//
//TITLE:        PLC: System informations
//
//              PLC: Systeminformationen
//
//
//--------------------------------------------------------------------------------
//
//IDENT:        AUTHOR:             DEPT:                              DATE:
//
//STD_DB050.1.1 Ph. Engler          MU664                              21-Dec-2000
//              ColdStart signals and counter integrated
//STD_DB050.1A  Ph. Engler          MU664                              05-Jan-2000
//              1st Release
//
//--------------------------------------------------------------------------------
//
//PURPOSE:  
//MANUAL : 
//CODE   :
//RESTRICTIONS:
//
//--------------------------------------------------------------------------------
//
//
//
//
//
//
//
AUTHOR : PE
FAMILY : GEN
NAME : SystemDB
VERSION : 9.9
  STRUCT
   Spare00 : WORD ;
   Startup : STRUCT
    CmdNewstartMan : BOOL ;	//Manual newstart active
    CmdNewstartAuto : BOOL ;	//Automatic newstart active
    CmdRestartMan : BOOL ;	//Manual restart requested
    CmdRestartAuto : BOOL ;	//Automatic restart requested
    CmdColdstartMan : BOOL ;	//Manual coldstart requested
    CmdColdstartAuto : BOOL ;	//Automatic coldstart requested
    NotUsed06 : BOOL ;
    NotUsed07 : BOOL ;
    CmdStartTestMode : BOOL ;	//Starts the test mode
   END_STRUCT ;
   StartupCounter : STRUCT
    NewstartMan : INT ;	//Number of manual newstart startups
    NewstartAuto : INT ;	//Number of automatic newstart startups
    RestartMan : INT ;	//Number of manual restart startups
    RestartAuto : INT ;	//Number of automatic restart startups
    ColdstartMan : INT ;	//Number of manual coldstart startups
    ColdstartAuto : INT ;	//Number of automatic coldstart startups
    NotUsed07 : INT ;
    NotUsed08 : INT ;
    NotUsed09 : INT ;
    NotUsed10 : INT ;
    NotUsed11 : INT ;
    NotUsed12 : INT ;
   END_STRUCT ;
   Hardware : STRUCT
    PLCBatteryFailure : BOOL ;
    NotUsed09 : BOOL ;
    NotUsed10 : BOOL ;
    NotUsed11 : BOOL ;
    NotUsed12 : BOOL ;
    NotUsed13 : BOOL ;
    NotUsed14 : BOOL ;
    NotUsed15 : BOOL ;
    VoltageOk : BOOL ;	//Control voltage ok
    EsGeneralOk : BOOL ;	//General emergency stop ok
    PowerOk : BOOL ;	//Power supply motor contactor panels ok
    FuseOk : BOOL ;	//Mini circuit breakers ok
    PlcOk : BOOL ;	//PLC ok
    FireOk : BOOL ;	//No fire alarms
    SmokeOk : BOOL ;	//No smoke alarms
    ExflapsOk : BOOL ;	//Explosion flaps ok
   END_STRUCT ;
   HardwareStop : STRUCT
    NotUsed08 : BOOL ;
    NotUsed09 : BOOL ;
    NotUsed10 : BOOL ;
    NotUsed11 : BOOL ;
    NotUsed12 : BOOL ;
    NotUsed13 : BOOL ;
    NotUsed14 : BOOL ;
    NotUsed15 : BOOL ;
    General : BOOL ;	//Stop from Hardware all circuits
    NotUsed01 : BOOL ;
    NotUsed02 : BOOL ;
    NotUsed03 : BOOL ;
    NotUsed04 : BOOL ;
    NotUsed05 : BOOL ;
    NotUsed06 : BOOL ;
    NotUsed07 : BOOL ;
   END_STRUCT ;
   GlobalFlags : STRUCT
    NotUsed08 : BOOL ;
    NotUsed09 : BOOL ;
    NotUsed10 : BOOL ;
    NotUsed11 : BOOL ;
    NotUsed12 : BOOL ;
    NotUsed13 : BOOL ;
    NotUsed14 : BOOL ;
    NotUsed15 : BOOL ;
    StaTest : BOOL ;	//Activates the test mode
    StaLOGOff : BOOL ;
    NotUsed02 : BOOL ;
    NotUsed03 : BOOL ;
    NotUsed04 : BOOL ;
    NotUsed05 : BOOL ;
    NotUsed06 : BOOL ;
    StaProtocolling : BOOL ;	//Activates the protocolling functionality of the elements
   END_STRUCT ;
   TestFunctions : STRUCT
    StaPLC1ComSimulation : BOOL ;
    StaPLC2ComSimulation : BOOL ;
    StaPLC3ComSimulation : BOOL ;
    StaPLC4ComSimulation : BOOL ;
    StaPLC5ComSimulation : BOOL ;
    StaPLC6ComSimulation : BOOL ;
    StaPLC7ComSimulation : BOOL ;
    StaPLC8ComSimulation : BOOL ;
    StaIOManager : BOOL ;	//IO's simulated with the IO-Manager
    StaHardware : BOOL ;	//IO's connected to the real hardware
    StaCWASimulation : BOOL ;	//CWA-Simulator on
    StaIOSimuli : BOOL ;	//IO's simulated with the IOSimuli
    StaDPSimulation : BOOL ;	//Simulation of DP-Scales
    StaWinAC : BOOL ;	//Testing on a WinAC
    NotUsed06 : BOOL ;
    StaPCDirectInhouseTest : BOOL ;	//Direct control channel for inhouse test
    StaPLC9ComSimulation : BOOL ;
    StaPLC10ComSimulation : BOOL ;
    StaPLC11ComSimulation : BOOL ;
    StaPLC12ComSimulation : BOOL ;
    StaPLC13ComSimulation : BOOL ;
    StaPLC14ComSimulation : BOOL ;
    StaPLC15ComSimulation : BOOL ;
    StaPLC16ComSimulation : BOOL ;
   END_STRUCT ;
   PlantID : STRUCT
    Product : ARRAY  [1 .. 15 ] OF //i.e. MELE_SMU01_99
    CHAR ;
    PlcNr : INT  := 1;
    GCSRelease : INT  := 2;
   END_STRUCT ;
  END_STRUCT ;	
BEGIN
   PlantID.Product[1] := 'M';
   PlantID.Product[2] := 'E';
   PlantID.Product[3] := 'L';
   PlantID.Product[4] := 'E';
   PlantID.Product[5] := '_';
   PlantID.Product[6] := 'S';
   PlantID.Product[7] := 'M';
   PlantID.Product[8] := 'U';
   PlantID.Product[9] := '0';
   PlantID.Product[10] := '1';
   PlantID.Product[11] := '_';
   PlantID.Product[12] := '9';
   PlantID.Product[13] := '9';
   PlantID.Product[14] := ' ';
   PlantID.Product[15] := ' ';
   PlantID.PlcNr := 1;
   PlantID.GCSRelease := 2;
END_DATA_BLOCK

DATA_BLOCK "PLC_DPInfo"	// DB 51
AUTHOR : SK
FAMILY : DP
NAME : DP_Diag
VERSION : 0.1
  STRUCT
   Master : ARRAY  [1 .. 4 ] OF STRUCT
    SlavesError : ARRAY  [1 .. 128 ] OF //List slaves with error
    BOOL ;
   END_STRUCT ;
  END_STRUCT ;	
BEGIN
END_DATA_BLOCK

DATA_BLOCK "SSA_SYS_ASI_Info"	// DB 52
AUTHOR : EA
FAMILY : GCS7LL
NAME : ASIInfo
VERSION : 0.1
  STRUCT
   Master : ARRAY  [1 .. 9 ] OF STRUCT
    Slaves_Faulted : STRUCT 	//1= Faulted Slaves A (Summery state)
     A : ARRAY  [0 .. 31 ] OF BOOL ;
     B : ARRAY  [0 .. 31 ] OF BOOL ;
    END_STRUCT ;
   END_STRUCT ;
  END_STRUCT ;	
BEGIN
END_DATA_BLOCK

DATA_BLOCK "SYS_DPInfoM1"	// DB 75
AUTHOR : SIEMENS
FAMILY : DP
VERSION : 0.0
"SYS_DP-Diagnosis"
BEGIN
END_DATA_BLOCK

DATA_BLOCK "SYS_DPInfoM2"	// DB 76
AUTHOR : SIEMENS
FAMILY : DP
VERSION : 0.0
"SYS_DP-Diagnosis"
BEGIN
END_DATA_BLOCK

DATA_BLOCK "SYS_DPInfoM3"	// DB 77
AUTHOR : SIEMENS
FAMILY : DP
VERSION : 0.0
"SYS_DP-Diagnosis"
BEGIN
END_DATA_BLOCK

DATA_BLOCK "SYS_DPInfoM4"	// DB 78
AUTHOR : SIEMENS
FAMILY : DP
VERSION : 0.0
"SYS_DP-Diagnosis"
BEGIN
END_DATA_BLOCK

DATA_BLOCK "PLC_BinListDB"	// DB 79
AUTHOR : EA
FAMILY : USW
VERSION : 0.0
"PLC_BinList"
BEGIN
END_DATA_BLOCK

DATA_BLOCK "SYS_SimpleDPInfo4DB"	// DB 98
AUTHOR : SK
FAMILY : DP
NAME : DP_Diag
VERSION : 0.1
  STRUCT
   tmpDataField : ARRAY  [1 .. 50 ] OF //Internal used (not relevant for user)
   BYTE ;
   Sum_SlavesNotPresent : INT ;	//Summary slaves not present
   List_SlavesNotPresent : ARRAY  [1 .. 128 ] OF //List slaves not present
   BOOL ;
   Sum_SlavesError : INT ;	//Summary slaves with error
   List_SlavesError : ARRAY  [1 .. 128 ] OF //List slaves with error
   BOOL ;
   OutRetVal : INT ;	//Error return value
   OutBusy : BOOL ;	//Diagnostic check active
  END_STRUCT ;	
BEGIN
END_DATA_BLOCK

DATA_BLOCK "SYS_StartWarningDB"	// DB 100
AUTHOR : EA
FAMILY : GCS7LL
VERSION : 0.0
"GCS7_StartWarning"
BEGIN
END_DATA_BLOCK

DATA_BLOCK "SSA_VIS_Filter"	// DB 2010
TITLE = PC Direct Control Interface General
//COPYRIGHT:    (C) 2000 BY  BUHLER LTD.
//                           CH-9240 UZWIL  SWITZERLAND
//
//PRODUCT:      SSA_VIS_Filter
//
//TITLE:        Filter Table for Viscontrol Status
//
//              Filter Table for Viscontrol Status
//
//
//--------------------------------------------------------------------------------
//
//IDENT:        AUTOR:              DEPT:                              DATE:
//
//SSW_DB003.1A  A.Egli              CT3                                01.Mrz.2003
//              1st Release 
//
//--------------------------------------------------------------------------------
//
//PURPOSE:      MANUAL : CTRxxMNA
//              CODE   : FC3
//
//RESTRICTIONS: S7
//              only for PC-Interface
//
//--------------------------------------------------------------------------------
//
//
//
VERSION : 0.0
  STRUCT
   ParBlockLen : INT  := 120;	//Block Lenght per Change bit as Bytes
   spare1 : WORD ;
   spare2 : WORD ;
   spare3 : WORD ;
   spare4 : WORD ;
   spare5 : WORD ;
   spare6 : WORD ;
   spare7 : WORD ;
   spare8 : WORD ;
   spare9 : WORD ;
   Filter : ARRAY  [123 .. 250 ] OF STRUCT
    Status0 : DWORD  := DW#16#C;
    Status1 : DWORD  := DW#16#10;
    Status2 : DWORD ;
    Status3 : DWORD  := DW#16#1023;
   END_STRUCT ;
  END_STRUCT ;	
BEGIN
   ParBlockLen := 120;
   spare3 := W#16#1404;
   Filter[123].Status0 := DW#16#C;
   Filter[123].Status1 := DW#16#10;
   Filter[123].Status3 := DW#16#1023;
   Filter[124].Status0 := DW#16#C;
   Filter[124].Status1 := DW#16#10;
   Filter[124].Status3 := DW#16#1023;
   Filter[125].Status0 := DW#16#C;
   Filter[125].Status1 := DW#16#10;
   Filter[125].Status3 := DW#16#1023;
   Filter[126].Status0 := DW#16#C;
   Filter[126].Status1 := DW#16#10;
   Filter[126].Status3 := DW#16#1023;
   Filter[127].Status0 := DW#16#C;
   Filter[127].Status1 := DW#16#10;
   Filter[127].Status3 := DW#16#1023;
   Filter[128].Status0 := DW#16#C;
   Filter[128].Status1 := DW#16#10;
   Filter[128].Status3 := DW#16#1023;
   Filter[129].Status0 := DW#16#C;
   Filter[129].Status1 := DW#16#10;
   Filter[129].Status3 := DW#16#1023;
   Filter[130].Status0 := DW#16#C;
   Filter[130].Status1 := DW#16#10;
   Filter[130].Status3 := DW#16#1023;
   Filter[131].Status0 := DW#16#C;
   Filter[131].Status1 := DW#16#10;
   Filter[131].Status3 := DW#16#1023;
   Filter[132].Status0 := DW#16#C;
   Filter[132].Status1 := DW#16#10;
   Filter[132].Status3 := DW#16#1023;
   Filter[133].Status0 := DW#16#C;
   Filter[133].Status1 := DW#16#10;
   Filter[133].Status3 := DW#16#1023;
   Filter[134].Status0 := DW#16#C;
   Filter[134].Status1 := DW#16#10;
   Filter[134].Status3 := DW#16#1023;
   Filter[135].Status0 := DW#16#C;
   Filter[135].Status1 := DW#16#10;
   Filter[135].Status3 := DW#16#1023;
   Filter[136].Status0 := DW#16#C;
   Filter[136].Status1 := DW#16#10;
   Filter[136].Status3 := DW#16#1023;
   Filter[137].Status0 := DW#16#C;
   Filter[137].Status1 := DW#16#10;
   Filter[137].Status3 := DW#16#1023;
   Filter[138].Status0 := DW#16#C;
   Filter[138].Status1 := DW#16#10;
   Filter[138].Status3 := DW#16#1023;
   Filter[139].Status0 := DW#16#C;
   Filter[139].Status1 := DW#16#10;
   Filter[139].Status3 := DW#16#1023;
   Filter[140].Status0 := DW#16#C;
   Filter[140].Status1 := DW#16#10;
   Filter[140].Status3 := DW#16#1023;
   Filter[141].Status0 := DW#16#C;
   Filter[141].Status1 := DW#16#10;
   Filter[141].Status3 := DW#16#1023;
   Filter[142].Status0 := DW#16#C;
   Filter[142].Status1 := DW#16#10;
   Filter[142].Status3 := DW#16#1023;
   Filter[143].Status0 := DW#16#C;
   Filter[143].Status1 := DW#16#10;
   Filter[143].Status3 := DW#16#1023;
   Filter[144].Status0 := DW#16#C;
   Filter[144].Status1 := DW#16#10;
   Filter[144].Status3 := DW#16#1023;
   Filter[145].Status0 := DW#16#C;
   Filter[145].Status1 := DW#16#10;
   Filter[145].Status3 := DW#16#1023;
   Filter[146].Status0 := DW#16#C;
   Filter[146].Status1 := DW#16#10;
   Filter[146].Status3 := DW#16#1023;
   Filter[147].Status0 := DW#16#C;
   Filter[147].Status1 := DW#16#10;
   Filter[147].Status3 := DW#16#1023;
   Filter[148].Status0 := DW#16#C;
   Filter[148].Status1 := DW#16#10;
   Filter[148].Status3 := DW#16#1023;
   Filter[149].Status0 := DW#16#C;
   Filter[149].Status1 := DW#16#10;
   Filter[149].Status3 := DW#16#1023;
   Filter[150].Status0 := DW#16#C;
   Filter[150].Status1 := DW#16#10;
   Filter[150].Status3 := DW#16#1023;
   Filter[151].Status0 := DW#16#C;
   Filter[151].Status1 := DW#16#10;
   Filter[151].Status3 := DW#16#1023;
   Filter[152].Status0 := DW#16#C;
   Filter[152].Status1 := DW#16#10;
   Filter[152].Status3 := DW#16#1023;
   Filter[153].Status0 := DW#16#C;
   Filter[153].Status1 := DW#16#10;
   Filter[153].Status3 := DW#16#1023;
   Filter[154].Status0 := DW#16#C;
   Filter[154].Status1 := DW#16#10;
   Filter[154].Status3 := DW#16#1023;
   Filter[155].Status0 := DW#16#C;
   Filter[155].Status1 := DW#16#10;
   Filter[155].Status3 := DW#16#1023;
   Filter[156].Status0 := DW#16#C;
   Filter[156].Status1 := DW#16#10;
   Filter[156].Status3 := DW#16#1023;
   Filter[157].Status0 := DW#16#C;
   Filter[157].Status1 := DW#16#10;
   Filter[157].Status3 := DW#16#1023;
   Filter[158].Status0 := DW#16#C;
   Filter[158].Status1 := DW#16#10;
   Filter[158].Status3 := DW#16#1023;
   Filter[159].Status0 := DW#16#C;
   Filter[159].Status1 := DW#16#10;
   Filter[159].Status3 := DW#16#1023;
   Filter[160].Status0 := DW#16#C;
   Filter[160].Status1 := DW#16#10;
   Filter[160].Status3 := DW#16#1023;
   Filter[161].Status0 := DW#16#C;
   Filter[161].Status1 := DW#16#10;
   Filter[161].Status3 := DW#16#1023;
   Filter[162].Status0 := DW#16#C;
   Filter[162].Status1 := DW#16#10;
   Filter[162].Status3 := DW#16#1023;
   Filter[163].Status0 := DW#16#C;
   Filter[163].Status1 := DW#16#10;
   Filter[163].Status3 := DW#16#1023;
   Filter[164].Status0 := DW#16#C;
   Filter[164].Status1 := DW#16#10;
   Filter[164].Status3 := DW#16#1023;
   Filter[165].Status0 := DW#16#C;
   Filter[165].Status1 := DW#16#10;
   Filter[165].Status3 := DW#16#1023;
   Filter[166].Status0 := DW#16#C;
   Filter[166].Status1 := DW#16#10;
   Filter[166].Status3 := DW#16#1023;
   Filter[167].Status0 := DW#16#C;
   Filter[167].Status1 := DW#16#10;
   Filter[167].Status3 := DW#16#1023;
   Filter[168].Status0 := DW#16#C;
   Filter[168].Status1 := DW#16#10;
   Filter[168].Status3 := DW#16#1023;
   Filter[169].Status0 := DW#16#C;
   Filter[169].Status1 := DW#16#10;
   Filter[169].Status3 := DW#16#1023;
   Filter[170].Status0 := DW#16#C;
   Filter[170].Status1 := DW#16#10;
   Filter[170].Status3 := DW#16#1023;
   Filter[171].Status0 := DW#16#C;
   Filter[171].Status1 := DW#16#10;
   Filter[171].Status3 := DW#16#1023;
   Filter[172].Status0 := DW#16#C;
   Filter[172].Status1 := DW#16#10;
   Filter[172].Status3 := DW#16#1023;
   Filter[173].Status0 := DW#16#C;
   Filter[173].Status1 := DW#16#10;
   Filter[173].Status3 := DW#16#1023;
   Filter[174].Status0 := DW#16#C;
   Filter[174].Status1 := DW#16#10;
   Filter[174].Status3 := DW#16#1023;
   Filter[175].Status0 := DW#16#C;
   Filter[175].Status1 := DW#16#10;
   Filter[175].Status3 := DW#16#1023;
   Filter[176].Status0 := DW#16#C;
   Filter[176].Status1 := DW#16#10;
   Filter[176].Status3 := DW#16#1023;
   Filter[177].Status0 := DW#16#C;
   Filter[177].Status1 := DW#16#10;
   Filter[177].Status3 := DW#16#1023;
   Filter[178].Status0 := DW#16#C;
   Filter[178].Status1 := DW#16#10;
   Filter[178].Status3 := DW#16#1023;
   Filter[179].Status0 := DW#16#C;
   Filter[179].Status1 := DW#16#10;
   Filter[179].Status3 := DW#16#1023;
   Filter[180].Status0 := DW#16#C;
   Filter[180].Status1 := DW#16#10;
   Filter[180].Status3 := DW#16#1023;
   Filter[181].Status0 := DW#16#C;
   Filter[181].Status1 := DW#16#10;
   Filter[181].Status3 := DW#16#1023;
   Filter[182].Status0 := DW#16#C;
   Filter[182].Status1 := DW#16#10;
   Filter[182].Status3 := DW#16#1023;
   Filter[183].Status0 := DW#16#C;
   Filter[183].Status1 := DW#16#10;
   Filter[183].Status3 := DW#16#1023;
   Filter[184].Status0 := DW#16#C;
   Filter[184].Status1 := DW#16#10;
   Filter[184].Status3 := DW#16#1023;
   Filter[185].Status0 := DW#16#C;
   Filter[185].Status1 := DW#16#10;
   Filter[185].Status3 := DW#16#1023;
   Filter[186].Status0 := DW#16#C;
   Filter[186].Status1 := DW#16#10;
   Filter[186].Status3 := DW#16#1023;
   Filter[187].Status0 := DW#16#C;
   Filter[187].Status1 := DW#16#10;
   Filter[187].Status3 := DW#16#1023;
   Filter[188].Status0 := DW#16#C;
   Filter[188].Status1 := DW#16#10;
   Filter[188].Status3 := DW#16#1023;
   Filter[189].Status0 := DW#16#C;
   Filter[189].Status1 := DW#16#10;
   Filter[189].Status3 := DW#16#1023;
   Filter[190].Status0 := DW#16#C;
   Filter[190].Status1 := DW#16#10;
   Filter[190].Status3 := DW#16#1023;
   Filter[191].Status0 := DW#16#C;
   Filter[191].Status1 := DW#16#10;
   Filter[191].Status3 := DW#16#1023;
   Filter[192].Status0 := DW#16#C;
   Filter[192].Status1 := DW#16#10;
   Filter[192].Status3 := DW#16#1023;
   Filter[193].Status0 := DW#16#C;
   Filter[193].Status1 := DW#16#10;
   Filter[193].Status3 := DW#16#1023;
   Filter[194].Status0 := DW#16#C;
   Filter[194].Status1 := DW#16#10;
   Filter[194].Status3 := DW#16#1023;
   Filter[195].Status0 := DW#16#C;
   Filter[195].Status1 := DW#16#10;
   Filter[195].Status3 := DW#16#1023;
   Filter[196].Status0 := DW#16#C;
   Filter[196].Status1 := DW#16#10;
   Filter[196].Status3 := DW#16#1023;
   Filter[197].Status0 := DW#16#C;
   Filter[197].Status1 := DW#16#10;
   Filter[197].Status3 := DW#16#1023;
   Filter[198].Status0 := DW#16#C;
   Filter[198].Status1 := DW#16#10;
   Filter[198].Status3 := DW#16#1023;
   Filter[199].Status0 := DW#16#C;
   Filter[199].Status1 := DW#16#10;
   Filter[199].Status3 := DW#16#1023;
   Filter[200].Status0 := DW#16#C;
   Filter[200].Status1 := DW#16#10;
   Filter[200].Status3 := DW#16#1023;
   Filter[201].Status0 := DW#16#C;
   Filter[201].Status1 := DW#16#10;
   Filter[201].Status3 := DW#16#1023;
   Filter[202].Status0 := DW#16#C;
   Filter[202].Status1 := DW#16#10;
   Filter[202].Status3 := DW#16#1023;
   Filter[203].Status0 := DW#16#C;
   Filter[203].Status1 := DW#16#10;
   Filter[203].Status3 := DW#16#1023;
   Filter[204].Status0 := DW#16#C;
   Filter[204].Status1 := DW#16#10;
   Filter[204].Status3 := DW#16#1023;
   Filter[205].Status0 := DW#16#C;
   Filter[205].Status1 := DW#16#10;
   Filter[205].Status3 := DW#16#1023;
   Filter[206].Status0 := DW#16#C;
   Filter[206].Status1 := DW#16#10;
   Filter[206].Status3 := DW#16#1023;
   Filter[207].Status0 := DW#16#C;
   Filter[207].Status1 := DW#16#10;
   Filter[207].Status3 := DW#16#1023;
   Filter[208].Status0 := DW#16#C;
   Filter[208].Status1 := DW#16#10;
   Filter[208].Status3 := DW#16#1023;
   Filter[209].Status0 := DW#16#C;
   Filter[209].Status1 := DW#16#10;
   Filter[209].Status3 := DW#16#1023;
   Filter[210].Status0 := DW#16#C;
   Filter[210].Status1 := DW#16#10;
   Filter[210].Status3 := DW#16#1023;
   Filter[211].Status0 := DW#16#C;
   Filter[211].Status1 := DW#16#10;
   Filter[211].Status3 := DW#16#1023;
   Filter[212].Status0 := DW#16#C;
   Filter[212].Status1 := DW#16#10;
   Filter[212].Status3 := DW#16#1023;
   Filter[213].Status0 := DW#16#C;
   Filter[213].Status1 := DW#16#10;
   Filter[213].Status3 := DW#16#1023;
   Filter[214].Status0 := DW#16#C;
   Filter[214].Status1 := DW#16#1;
   Filter[214].Status2 := DW#16#10;
   Filter[214].Status3 := DW#16#100002;
   Filter[215].Status0 := DW#16#C;
   Filter[215].Status1 := DW#16#10;
   Filter[215].Status3 := DW#16#1023;
   Filter[216].Status0 := DW#16#C;
   Filter[216].Status1 := DW#16#10;
   Filter[216].Status3 := DW#16#1023;
   Filter[217].Status0 := DW#16#C;
   Filter[217].Status1 := DW#16#10;
   Filter[217].Status3 := DW#16#1023;
   Filter[218].Status0 := DW#16#C;
   Filter[218].Status1 := DW#16#10;
   Filter[218].Status3 := DW#16#1023;
   Filter[219].Status0 := DW#16#C;
   Filter[219].Status1 := DW#16#10;
   Filter[219].Status3 := DW#16#1023;
   Filter[220].Status0 := DW#16#C;
   Filter[220].Status1 := DW#16#10;
   Filter[220].Status3 := DW#16#1023;
   Filter[221].Status0 := DW#16#C;
   Filter[221].Status1 := DW#16#10;
   Filter[221].Status3 := DW#16#1023;
   Filter[222].Status0 := DW#16#C;
   Filter[222].Status1 := DW#16#10;
   Filter[222].Status3 := DW#16#1023;
   Filter[223].Status0 := DW#16#C;
   Filter[223].Status1 := DW#16#10;
   Filter[223].Status3 := DW#16#1023;
   Filter[224].Status0 := DW#16#C;
   Filter[224].Status1 := DW#16#10;
   Filter[224].Status3 := DW#16#1023;
   Filter[225].Status0 := DW#16#C;
   Filter[225].Status1 := DW#16#10;
   Filter[225].Status3 := DW#16#1023;
   Filter[226].Status0 := DW#16#C;
   Filter[226].Status1 := DW#16#10;
   Filter[226].Status3 := DW#16#1023;
   Filter[227].Status0 := DW#16#C;
   Filter[227].Status1 := DW#16#10;
   Filter[227].Status3 := DW#16#1023;
   Filter[228].Status0 := DW#16#C;
   Filter[228].Status1 := DW#16#10;
   Filter[228].Status3 := DW#16#1023;
   Filter[229].Status0 := DW#16#C;
   Filter[229].Status1 := DW#16#10;
   Filter[229].Status3 := DW#16#1023;
   Filter[230].Status0 := DW#16#C;
   Filter[230].Status1 := DW#16#10;
   Filter[230].Status3 := DW#16#1023;
   Filter[231].Status0 := DW#16#C;
   Filter[231].Status1 := DW#16#10;
   Filter[231].Status3 := DW#16#1023;
   Filter[232].Status0 := DW#16#C;
   Filter[232].Status1 := DW#16#10;
   Filter[232].Status3 := DW#16#1023;
   Filter[233].Status0 := DW#16#C;
   Filter[233].Status1 := DW#16#10;
   Filter[233].Status3 := DW#16#1023;
   Filter[234].Status0 := DW#16#C;
   Filter[234].Status1 := DW#16#10;
   Filter[234].Status3 := DW#16#1023;
   Filter[235].Status0 := DW#16#C;
   Filter[235].Status1 := DW#16#10;
   Filter[235].Status3 := DW#16#1023;
   Filter[236].Status0 := DW#16#C;
   Filter[236].Status1 := DW#16#10;
   Filter[236].Status3 := DW#16#1023;
   Filter[237].Status0 := DW#16#C;
   Filter[237].Status1 := DW#16#10;
   Filter[237].Status3 := DW#16#1023;
   Filter[238].Status0 := DW#16#C;
   Filter[238].Status1 := DW#16#10;
   Filter[238].Status3 := DW#16#1023;
   Filter[239].Status0 := DW#16#C;
   Filter[239].Status1 := DW#16#10;
   Filter[239].Status3 := DW#16#1023;
   Filter[240].Status0 := DW#16#C;
   Filter[240].Status1 := DW#16#10;
   Filter[240].Status3 := DW#16#1023;
   Filter[241].Status0 := DW#16#C;
   Filter[241].Status1 := DW#16#10;
   Filter[241].Status3 := DW#16#1023;
   Filter[242].Status0 := DW#16#C;
   Filter[242].Status1 := DW#16#10;
   Filter[242].Status3 := DW#16#1023;
   Filter[243].Status0 := DW#16#C;
   Filter[243].Status1 := DW#16#10;
   Filter[243].Status3 := DW#16#1023;
   Filter[244].Status0 := DW#16#C;
   Filter[244].Status1 := DW#16#10;
   Filter[244].Status3 := DW#16#1023;
   Filter[245].Status0 := DW#16#C;
   Filter[245].Status1 := DW#16#10;
   Filter[245].Status3 := DW#16#1023;
   Filter[246].Status0 := DW#16#C;
   Filter[246].Status1 := DW#16#10;
   Filter[246].Status3 := DW#16#1023;
   Filter[247].Status0 := DW#16#C;
   Filter[247].Status1 := DW#16#10;
   Filter[247].Status3 := DW#16#1023;
   Filter[248].Status0 := DW#16#C;
   Filter[248].Status1 := DW#16#10;
   Filter[248].Status3 := DW#16#1023;
   Filter[249].Status0 := DW#16#C;
   Filter[249].Status1 := DW#16#10;
   Filter[249].Status3 := DW#16#1023;
   Filter[250].Status0 := DW#16#C;
   Filter[250].Status1 := DW#16#10;
   Filter[250].Status3 := DW#16#1023;
END_DATA_BLOCK

ORGANIZATION_BLOCK "SYS_MainProgram"	// OB 1
AUTHOR : ASW
FAMILY : SYS
NAME : MainProg
VERSION : 0.1
VAR_TEMP
  OB1_EV_CLASS : BYTE ;	//Bits 0-3 = 1 (Coming event), Bits 4-7 = 1 (Event class 1)
  OB1_SCAN_1 : BYTE ;	//1 (Cold restart scan 1 of OB 1), 3 (Scan 2-n of OB 1)
  OB1_PRIORITY : BYTE ;	//1 (Priority of 1 is lowest)
  OB1_OB_NUMBR : BYTE ;	//1 (Organization block 1, OB1)
  OB1_RESERVED_1 : BYTE ;	//Reserved for system
  OB1_RESERVED_2 : BYTE ;	//Reserved for system
  OB1_PREV_CYCLE : INT ;	//Cycle time of previous OB1 scan (milliseconds)
  OB1_MIN_CYCLE : INT ;	//Minimum cycle time of OB1 (milliseconds)
  OB1_MAX_CYCLE : INT ;	//Maximum cycle time of OB1 (milliseconds)
  OB1_DATE_TIME : DATE_AND_TIME ;	//Date and time OB1 started
END_VAR
BEGIN
NETWORK
TITLE = Timer Flag
      CALL  "SYS_InitFlagTimer";
NETWORK
TITLE = Call IO-Simulation
      UC    "TEST_IOSIMULI_Copy";
NETWORK
TITLE = Call Group
      UC    "SYS_CallGroup";
NETWORK
TITLE = Call Line
NETWORK
TITLE = Call CBIT
NETWORK
TITLE = Detailed Diagnosis in OB82 (interrupt)
      CALL  "SYS_DPDiagMain";
NETWORK
TITLE = Reset startup flags
      SET;
      R     "PLC_SystemDB".Startup.CmdRestartMan;
      R     "PLC_SystemDB".Startup.CmdRestartAuto;
NETWORK
TITLE = End of block
      BE;
END_ORGANIZATION_BLOCK

ORGANIZATION_BLOCK "SYS_CYCL_FLT"	// OB 80
TITLE = "Cycle Time Fault"
//COPYRIGHT:    (C) 2000 BY  BUHLER AG
//                           CH-9240 UZWIL  SWITZERLAND
//
//PRODUCT:      PROJECT
//
//TITLE:        Time Error Organization Block (OB80)
//
//--------------------------------------------------------------------------------
//IDENT:        AUTHOR:             DEPT:                             DATE:
//
//STD_OB80.2.0  A.Egli              CT3                               12-Jul-2004
//              Log message added
//
//--------------------------------------------------------------------------------
//
//PURPOSE:      
//
//RESTRICTIONS: 
//
//--------------------------------------------------------------------------------
//
AUTHOR : EA
FAMILY : ASW
NAME : CYCL_FLT
VERSION : 2.0
VAR_TEMP
  OB80_EV_CLASS : BYTE ;	//16#35, Event class 3, Entering event state, Internal fault event
  OB80_FLT_ID : BYTE ;	//16#XX, Fault identifcation code
  OB80_PRIORITY : BYTE ;	//26 (Priority of 1 is lowest)
  OB80_OB_NUMBR : BYTE ;	//80 (Organization block 80, OB80)
  OB80_RESERVED_1 : BYTE ;	//Reserved for system
  OB80_RESERVED_2 : BYTE ;	//Reserved for system
  OB80_ERROR_INFO : WORD ;	//Error information on event
  OB80_ERR_EV_CLASS : BYTE ;	//Class of event causing error
  OB80_ERR_EV_NUM : BYTE ;	//Number of event causing error
  OB80_OB_PRIORITY : BYTE ;	//Priority of OB causing error
  OB80_OB_NUM : BYTE ;	//Number of OB causing error
  OB80_DATE_TIME : DATE_AND_TIME ;	//Date and time OB80 started
  tmpHeader : WORD ;
  tmpObjNo : WORD ;	//OB-Nummer [80..121]
  EVClass_FLTID : WORD ;	//EV_Class / FLT_ID
  tmpPara3 : WORD ;	//Reserved 1 for system
  tmpYearMonth : WORD ;
  tmpDayHour : WORD ;
  tmpMinSec : WORD ;
  tmpNoStop : BOOL ;
END_VAR
BEGIN
NETWORK
TITLE =
NETWORK
TITLE = Log Message: Header
      A(;
      L     #OB80_EV_CLASS;
      L     B#16#38;	// going
      ==I;
      );
      JCN   komm;
      L     3;
      JU    tran;
komm: L     1;	// coming
tran: SLW   5;
      +     11;	// NEW MessageFormatNo
      T     #tmpHeader;
NETWORK
TITLE = Log Message: Para1 = Object Number
//--System Message---
      L     80;
      T     #tmpObjNo;
NETWORK
TITLE = Log Message: Para2 to 11
////
//Para2: EV_Class / FLT_ID
      L     #OB80_FLT_ID;
      L     W#16#FF;	// Only Low Byte
      AW;
      L     #OB80_EV_CLASS;
      SLD   8;
      OW;
      T     #EVClass_FLTID;
//Para3: Depending on fault identification code
      L     #OB80_OB_NUMBR;
      T     #tmpPara3;
//Para9 to 11: Date/Time
      LAR1  P##OB80_DATE_TIME;
      L     LB [AR1,P#0.0];
      BTI;
      SLD   8;
      L     LB [AR1,P#1.0];
      BTI;
      OW;
      T     #tmpYearMonth;
      L     LB [AR1,P#2.0];
      BTI;
      SLD   8;
      L     LB [AR1,P#3.0];
      BTI;
      OW;
      T     #tmpDayHour;
      L     LB [AR1,P#4.0];
      BTI;
      SLD   8;
      L     LB [AR1,P#5.0];
      BTI;
      OW;
      T     #tmpMinSec;
NETWORK
TITLE = Faults without STOP
//// alle auskommentierten Einträge führen in STOP
      CLR;	//init.VKE  
// 1 Cycle time exceeded
//      O(    
//      L     #OB80_FLT_ID
//      L     B#16#1                      // 
//      ==I   
//      )     
// 2 Called OB is still being executed
//      O(    
//      L     #OB80_FLT_ID
//      L     B#16#2                      // 
//      ==I   
//      )     
// 5 Elapsed time-of-day interrupt due to moving the clock forwar
//      O(    
//      L     #OB80_FLT_ID
//      L     B#16#5                      // 
//      ==I   
//      )     
// 6 Elapsed time-of-day interrupt on return to RUN after HOLD
//      O(    
//      L     #OB80_FLT_ID
//      L     B#16#6                      // 
//      ==I   
//      )     
// 7 Overflow of OB request buffer
//      O(    
//      L     #OB80_FLT_ID
//      L     B#16#26                     // 
//      ==I   
//      )     
      =     #tmpNoStop;
NETWORK
TITLE = Log Message: Entry
//Entre Log Message
      AN    #tmpNoStop;
      S     "SYS_LOG_Queue".CmdAddFastMsg;
      CALL  "SYS_LOG_EntryQueue" (
           DBNumber                 := 5,
           Header                   := #tmpHeader,
           Para1                    := #tmpObjNo,
           Para2                    := #EVClass_FLTID,
           Para3                    := #tmpPara3,
           Para4                    := W#16#0,
           Para5                    := W#16#0,
           Para6                    := W#16#0,
           Para7                    := W#16#0,
           Para8                    := W#16#0,
           Para9                    := #tmpYearMonth,
           Para10                   := #tmpDayHour,
           Para11                   := #tmpMinSec);	//Header / Para1: ObjectNo / Para2: Class / FLTID / Para3: OB Number / Para9:  Year / Month / Para10: Day  / Hour / Para11: Min  / Sec 
NETWORK
TITLE = Stop PLC
      A     #tmpNoStop;
      BEC;
//**********************
// Bring CPU to Stop
      CALL  "SIEMENS_STP";
//**********************
END_ORGANIZATION_BLOCK

ORGANIZATION_BLOCK "SYS_PS_FLT"	// OB 81
TITLE = "Power Supply Fault"
//COPYRIGHT:    (C) 2000 BY  BUHLER AG
//                           CH-9240 UZWIL  SWITZERLAND
//
//PRODUCT:      Project
//
//TITLE:        Power supply fault
//               Batterie monitoring
//              Stromversorgungsfehler
//               Batterieüberwachung              
//
//--------------------------------------------------------------------------------
//IDENT:        AUTHOR:             DEPT:                              DATE:
//
//Pxx_OB081.1.1 Ph. Engler          MU664                              12-Feb-2003
//              Redesign GCS7 Release 2
//Pxx_OB081.1.0 Ph. Engler          MU664                              29-Mar-2001
//              1st Release
//
//--------------------------------------------------------------------------------
//
//PURPOSE:      
//
//RESTRICTIONS: 
//
//--------------------------------------------------------------------------------
//
AUTHOR : PE
FAMILY : ASW
NAME : PS_FLT
VERSION : 2.0
VAR_TEMP
  OB81_EV_CLASS : BYTE ;	//16#39, Event class 3, Entering event state, Internal fault event
  OB81_FLT_ID : BYTE ;	//16#XX, Fault identification code
  OB81_PRIORITY : BYTE ;	//26/28 (Priority of 1 is lowest)
  OB81_OB_NUMBR : BYTE ;	//81 (Organization block 81, OB81)
  OB81_RESERVED_1 : BYTE ;	//Reserved for system
  OB81_RESERVED_2 : BYTE ;	//Reserved for system
  OB81_MDL_ADDR : INT ;	//Reserved for system
  OB81_RESERVED_3 : BYTE ;	//Reserved for system
  OB81_RESERVED_4 : BYTE ;	//Reserved for system
  OB81_RESERVED_5 : BYTE ;	//Reserved for system
  OB81_RESERVED_6 : BYTE ;	//Reserved for system
  OB81_DATE_TIME : DATE_AND_TIME ;	//Date and time OB81 started
  tmpHeader : WORD ;
  tmpObjNo : WORD ;	//OB-Nummer [80..121]
  EVClass_FLTID : WORD ;	//EV_Class / FLT_ID
  tmpPara3 : WORD ;
  tmpYearMonth : WORD ;
  tmpDayHour : WORD ;
  tmpMinSec : WORD ;
  tmpNoStop : BOOL ;
END_VAR
BEGIN
NETWORK
TITLE = EC Event class
      L     #OB81_EV_CLASS;
      L     B#16#39;	// CONST.event_failure
      ==I;
      JC    FAIL;
      L     #OB81_EV_CLASS;
      L     B#16#38;	// CONST.event_failure_reset
      ==I;
      JC    FRES;
      BEU;
NETWORK
TITLE = EF EVENT_FAILURE
FAIL: NOP   0;
      L     #OB81_FLT_ID;
      L     B#16#21;	// Battery failure
      ==I;
      JCN   EF01;
      S     "PLC_SystemDB".Hardware.PLCBatteryFailure;
      JU    LOG;
EF01: NOP   0;
      JU    LOG;
NETWORK
TITLE = ER EVENT_FAILURE_RESET
FRES: NOP   0;
      L     #OB81_FLT_ID;
      L     B#16#21;	// Battery failure
      ==I;
      JCN   ER01;
      R     "PLC_SystemDB".Hardware.PLCBatteryFailure;
      JU    LOG;
ER01: NOP   0;
      JU    LOG;
NETWORK
TITLE = Log Message: Header
LOG:  A(;
      L     #OB81_EV_CLASS;
      L     B#16#38;	// going
      ==I;
      );
      JCN   komm;
      L     3;
      JU    tran;
komm: L     1;	// coming
tran: SLW   5;
      +     11;	// NEW MessageFormatNo
      T     #tmpHeader;
NETWORK
TITLE = Log Message: Para1 = Object Number
//--System Message---
      L     #OB81_OB_NUMBR;
      T     #tmpObjNo;
NETWORK
TITLE = Log Message: Para2 to 11
////
//Para2: EV_Class / FLT_ID
      L     #OB81_FLT_ID;
      L     W#16#FF;	// Only Low Byte
      AW;
      L     #OB81_EV_CLASS;
      SLD   8;
      OW;
      T     #EVClass_FLTID;
//Para3: Depending on fault identification code
      L     #OB81_OB_NUMBR;
      T     #tmpPara3;
//Para9 to 11: Date/Time
      LAR1  P##OB81_DATE_TIME;
      L     LB [AR1,P#0.0];
      BTI;
      SLD   8;
      L     LB [AR1,P#1.0];
      BTI;
      OW;
      T     #tmpYearMonth;
      L     LB [AR1,P#2.0];
      BTI;
      SLD   8;
      L     LB [AR1,P#3.0];
      BTI;
      OW;
      T     #tmpDayHour;
      L     LB [AR1,P#4.0];
      BTI;
      SLD   8;
      L     LB [AR1,P#5.0];
      BTI;
      OW;
      T     #tmpMinSec;
NETWORK
TITLE = Log Message: Entry
//Entre Log Message
      CALL  "SYS_LOG_EntryQueue" (
           DBNumber                 := 5,
           Header                   := #tmpHeader,
           Para1                    := #tmpObjNo,
           Para2                    := #EVClass_FLTID,
           Para3                    := #tmpPara3,
           Para4                    := W#16#0,
           Para5                    := W#16#0,
           Para6                    := W#16#0,
           Para7                    := W#16#0,
           Para8                    := W#16#0,
           Para9                    := #tmpYearMonth,
           Para10                   := #tmpDayHour,
           Para11                   := #tmpMinSec);	//Header / Para1: ObjectNo / Para2: Class / FLTID / Para3: OB Number / Para9:  Year / Month / Para10: Day  / Hour / Para11: Min  / Sec 
NETWORK
TITLE = End of block
      BE;
END_ORGANIZATION_BLOCK

ORGANIZATION_BLOCK "SYS_IO_FLT1"	// OB 82
TITLE = "I/O Point Fault"
//COPYRIGHT:    (C) 2000 BY  BUHLER AG
//                           CH-9240 UZWIL  SWITZERLAND
//
//PRODUCT:      PROJECT
//
//TITLE:        Diagnostic Alarm
//
//--------------------------------------------------------------------------------
//IDENT:        AUTHOR:             DEPT:                             DATE:
//
//OB082.2.0     A.Egli              CT3                               14-Jul-2004
//              Log message added
//OB082.1.0     Ph. Engler          MU664                             10-Feb-2003
//              Redesign GCS7 Release 2
//
//--------------------------------------------------------------------------------
//
//PURPOSE:      
//
//RESTRICTIONS: 
//
//--------------------------------------------------------------------------------
//
AUTHOR : EA
FAMILY : ASW
NAME : IOFLT1
VERSION : 2.0
VAR_TEMP
  OB82_EV_CLASS : BYTE ;	//16#39, Event class 3, Entering event state, Internal fault event
  OB82_FLT_ID : BYTE ;	//16#XX, Fault identifcation code
  OB82_PRIORITY : BYTE ;	//26/28 (Priority of 1 is lowest)
  OB82_OB_NUMBR : BYTE ;	//82 (Organization block 82, OB82)
  OB82_RESERVED_1 : BYTE ;	//Reserved for system
  OB82_IO_FLAG : BYTE ;	//Input (01010100), Output (01010101)
  OB82_MDL_ADDR : INT ;	//Base address of module with fault
  OB82_MDL_DEFECT : BOOL ;	//Module defective
  OB82_INT_FAULT : BOOL ;	//Internal fault
  OB82_EXT_FAULT : BOOL ;	//External fault
  OB82_PNT_INFO : BOOL ;	//Point information
  OB82_EXT_VOLTAGE : BOOL ;	//External voltage low
  OB82_FLD_CONNCTR : BOOL ;	//Field wiring connector missing
  OB82_NO_CONFIG : BOOL ;	//Module has no configuration data
  OB82_CONFIG_ERR : BOOL ;	//Module has configuration error
  OB82_MDL_TYPE : BYTE ;	//Type of module
  OB82_SUB_NDL_ERR : BOOL ;	//Sub-Module is missing or has error
  OB82_COMM_FAULT : BOOL ;	//Communication fault
  OB82_MDL_STOP : BOOL ;	//Module is stopped
  OB82_WTCH_DOG_FLT : BOOL ;	//Watch dog timer stopped module
  OB82_INT_PS_FLT : BOOL ;	//Internal power supply fault
  OB82_PRIM_BATT_FLT : BOOL ;	//Primary battery is in fault
  OB82_BCKUP_BATT_FLT : BOOL ;	//Backup battery is in fault
  OB82_RESERVED_2 : BOOL ;	//Reserved for system
  OB82_RACK_FLT : BOOL ;	//Rack fault, only for bus interface module
  OB82_PROC_FLT : BOOL ;	//Processor fault
  OB82_EPROM_FLT : BOOL ;	//EPROM fault
  OB82_RAM_FLT : BOOL ;	//RAM fault
  OB82_ADU_FLT : BOOL ;	//ADU fault
  OB82_FUSE_FLT : BOOL ;	//Fuse fault
  OB82_HW_INTR_FLT : BOOL ;	//Hardware interupt input in fault
  OB82_RESERVED_3 : BOOL ;	//Reserved for system
  OB82_DATE_TIME : DATE_AND_TIME ;	//Date and time OB82 started
  tmpHeader : WORD ;
  tmpObjNo : WORD ;	//OB-Nummer [80..121]
  EVClass_FLTID : WORD ;	//EV_Class / FLT_ID
  tmpPara3 : WORD ;	//Reserved 1 for system
  tmpPara4 : WORD ;	//Input module (01010100), Output module (01010101)
  tmpPara5 : WORD ;	//Base address of module with point fault
  tmpPara6 : WORD ;	//Module type with point fault
  tmpYearMonth : WORD ;
  tmpDayHour : WORD ;
  tmpMinSec : WORD ;
  tmpNoStop : BOOL ;
END_VAR
BEGIN
NETWORK
TITLE = Detailed Diagnosis in OB82 (interrupt)
      CALL  "SYS_DPDiagMain";
NETWORK
TITLE = Log Message: Header
      A(;
      L     #OB82_EV_CLASS;
      L     B#16#38;	// going
      ==I;
      );
      JCN   komm;
      L     3;
      JU    tran;
komm: L     1;	// coming
tran: SLW   5;
      +     11;	// NEW MessageFormatNo
      T     #tmpHeader;
NETWORK
TITLE = Log Message: Para1 = Object Number
//--System Message---
      L     82;
      T     #tmpObjNo;
NETWORK
TITLE = Log Message: Para2 to 11
////
//Para2: EV_Class / FLT_ID
      L     #OB82_FLT_ID;
      L     W#16#FF;	// Only Low Byte
      AW;
      L     #OB82_EV_CLASS;
      SLD   8;
      OW;
      T     #EVClass_FLTID;
//Para3: Depending on fault identification code
      L     #OB82_OB_NUMBR;
      T     #tmpPara3;
//Para4: Input (01010100), Output (01010101)
      L     #OB82_IO_FLAG;
      T     #tmpPara4;
//Para5: Base address of module with fault
      L     #OB82_MDL_ADDR;
      T     #tmpPara5;
//Para6: Type of module
      L     #OB82_MDL_TYPE;
      T     #tmpPara6;
//Para9 to 11: Date/Time
      LAR1  P##OB82_DATE_TIME;
      L     LB [AR1,P#0.0];
      BTI;
      SLD   8;
      L     LB [AR1,P#1.0];
      BTI;
      OW;
      T     #tmpYearMonth;
      L     LB [AR1,P#2.0];
      BTI;
      SLD   8;
      L     LB [AR1,P#3.0];
      BTI;
      OW;
      T     #tmpDayHour;
      L     LB [AR1,P#4.0];
      BTI;
      SLD   8;
      L     LB [AR1,P#5.0];
      BTI;
      OW;
      T     #tmpMinSec;
NETWORK
TITLE = Faults without STOP
//// alle auskommentierten Einträge führen in STOP
      CLR;	//init.VKE  
// Diagnostic Alarm
      O(;
      L     #OB82_FLT_ID;
      L     B#16#42;	// 
      ==I;
      );
      =     #tmpNoStop;
NETWORK
TITLE = Log Message: Entry
//Entre Log Message
      AN    #tmpNoStop;
      S     "SYS_LOG_Queue".CmdAddFastMsg;
      CALL  "SYS_LOG_EntryQueue" (
           DBNumber                 := 5,
           Header                   := #tmpHeader,
           Para1                    := #tmpObjNo,
           Para2                    := #EVClass_FLTID,
           Para3                    := #tmpPara3,
           Para4                    := #tmpPara4,
           Para5                    := #tmpPara5,
           Para6                    := #tmpPara6,
           Para7                    := W#16#0,
           Para8                    := W#16#0,
           Para9                    := #tmpYearMonth,
           Para10                   := #tmpDayHour,
           Para11                   := #tmpMinSec);	//Header / Para1: ObjectNo / Para2: Class / FLTID / Para3: OB Number / OB82_MDL_ID / OB82_MDL_ADDR / OB82_MDL_TYPE / Para9:  Year / Month / Para10: Day  / Hour / Para11: Min  / Sec 
NETWORK
TITLE = Stop PLC
      A     #tmpNoStop;
      BEC;
//**********************
// Bring CPU to Stop
      CALL  "SIEMENS_STP";
//**********************
NETWORK
TITLE = End of block
      BE;
END_ORGANIZATION_BLOCK

ORGANIZATION_BLOCK "SYS_IO_FLT2"	// OB 83
TITLE = "I/O Point Fault"
//COPYRIGHT:    (C) 2000 BY  BUHLER AG
//                           CH-9240 UZWIL  SWITZERLAND
//
//PRODUCT:      PROJECT
//
//TITLE:        Insert / Remove Module Interrupt Organization Block (OB83)
//              
//
//--------------------------------------------------------------------------------
//IDENT:        AUTHOR:             DEPT:                             DATE:
//
//OB083.2.0     A.Egli              CT3                               26-Jul-2004
//              Log message added
//OB83.1B       Tho                 FU53                              16-Dez-99
//              FU-Version erstellt
//OB83.1A       TIK                 MU664                             13-Apr-99
//              1st Release
//--------------------------------------------------------------------------------
//
//PURPOSE:      
//
//RESTRICTIONS: 
//
//--------------------------------------------------------------------------------
//
AUTHOR : EA
FAMILY : ASW
NAME : IOFLT2
VERSION : 2.0
VAR_TEMP
  OB83_EV_CLASS : BYTE ;	//16#38/39, Event class 3, module inserted/removed (8/9)
  OB83_FLT_ID : BYTE ;	//16#XX, Fault identifcation code
  OB83_PRIORITY : BYTE ;	//26/28 (Priority of 1 is lowest)
  OB83_OB_NUMBR : BYTE ;	//83 (Organization block 83, OB83)
  OB83_RESERVED_1 : BYTE ;	//Reserved for system
  OB83_MDL_ID : BYTE ;	//Input module (01010100), Output module (01010101)
  OB83_MDL_ADDR : WORD ;	//Base address of module with point fault
  OB83_RACK_NUM : WORD ;	//Number of rack that has module with point fault
  OB83_MDL_TYPE : WORD ;	//Module type with point fault
  OB83_DATE_TIME : DATE_AND_TIME ;	//Date and time OB83 started
  tmpHeader : WORD ;
  tmpObjNo : WORD ;	//OB-Nummer [80..121]
  EVClass_FLTID : WORD ;	//EV_Class / FLT_ID
  tmpPara3 : WORD ;	//Reserved 1 for system
  tmpPara4 : WORD ;	//Input module (01010100), Output module (01010101)
  tmpPara5 : WORD ;	//Base address of module with point fault
  tmpPara6 : WORD ;	//Module type with point fault
  tmpYearMonth : WORD ;
  tmpDayHour : WORD ;
  tmpMinSec : WORD ;
  tmpNoStop : BOOL ;
END_VAR
BEGIN
NETWORK
TITLE =
NETWORK
TITLE = Log Message: Header
      A(;
      L     #OB83_EV_CLASS;
      L     B#16#38;	// going
      ==I;
      );
      JCN   komm;
      L     3;
      JU    tran;
komm: L     1;	// coming
tran: SLW   5;
      +     11;	// NEW MessageFormatNo
      T     #tmpHeader;
NETWORK
TITLE = Log Message: Para1 = Object Number
//--System Message---
      L     83;
      T     #tmpObjNo;
NETWORK
TITLE = Log Message: Para2 to 11
////
//Para2: EV_Class / FLT_ID
      L     #OB83_FLT_ID;
      L     W#16#FF;	// Only Low Byte
      AW;
      L     #OB83_EV_CLASS;
      SLD   8;
      OW;
      T     #EVClass_FLTID;
//Para3: Depending on fault identification code
      L     #OB83_OB_NUMBR;
      T     #tmpPara3;
//Para4: Input module (01010100), Output module (01010101)
      L     #OB83_MDL_ID;
      T     #tmpPara4;
//Para5: Base address of module with point fault
      L     #OB83_MDL_ADDR;
      T     #tmpPara5;
//Para6: Module type with point fault
      L     #OB83_MDL_TYPE;
      T     #tmpPara6;
//Para9 to 11: Date/Time
      LAR1  P##OB83_DATE_TIME;
      L     LB [AR1,P#0.0];
      BTI;
      SLD   8;
      L     LB [AR1,P#1.0];
      BTI;
      OW;
      T     #tmpYearMonth;
      L     LB [AR1,P#2.0];
      BTI;
      SLD   8;
      L     LB [AR1,P#3.0];
      BTI;
      OW;
      T     #tmpDayHour;
      L     LB [AR1,P#4.0];
      BTI;
      SLD   8;
      L     LB [AR1,P#5.0];
      BTI;
      OW;
      T     #tmpMinSec;
NETWORK
TITLE = Faults without STOP
//// alle auskommentierten Einträge führen in STOP
      CLR;
// 61 Module removed or not responding
//      O(    
//      L     #OB83_FLT_ID
//      L     B#16#61                     // 
//      ==I   
//      )     
// 63 Module inserted but incorrect module type
//      O(    
//      L     #OB83_FLT_ID
//      L     B#16#63                     // 
//      ==I   
//      )     
// 64 Module inserted but problem
//      O(    
//      L     #OB83_FLT_ID
//      L     B#16#64                     // 
//      ==I   
//      )     
// 65 Module inserted but error in module parameter assignment
//      O(    
//      L     #OB83_FLT_ID
//      L     B#16#65                     // 
//      ==I   
//      )     
      =     #tmpNoStop;
NETWORK
TITLE = Log Message: Entry
//Entre Log Message
      AN    #tmpNoStop;
      S     "SYS_LOG_Queue".CmdAddFastMsg;
      CALL  "SYS_LOG_EntryQueue" (
           DBNumber                 := 5,
           Header                   := #tmpHeader,
           Para1                    := #tmpObjNo,
           Para2                    := #EVClass_FLTID,
           Para3                    := #tmpPara3,
           Para4                    := #tmpPara4,
           Para5                    := #tmpPara5,
           Para6                    := #tmpPara6,
           Para7                    := W#16#0,
           Para8                    := W#16#0,
           Para9                    := #tmpYearMonth,
           Para10                   := #tmpDayHour,
           Para11                   := #tmpMinSec);	//Header / Para1: ObjectNo / Para2: Class / FLTID / Para3: OB Number / OB83_MDL_ID / OB83_MDL_ADDR / OB83_MDL_TYPE / Para9:  Year / Month / Para10: Day  / Hour / Para11: Min  / Sec 
NETWORK
TITLE = Stop PLC
      A     #tmpNoStop;
      BEC;
//**********************
// Bring CPU to Stop
      CALL  "SIEMENS_STP";
//**********************
NETWORK
TITLE = End of block
      BE;
END_ORGANIZATION_BLOCK

